// TIA Portal V19 export
FUNCTION "CEB_1" : Void   // FC14, LAD
{ S7_Optimized_Access := 'TRUE' }
// stored: SetENOAutomatically false
BEGIN

REGION Network 1: CEB_1 START
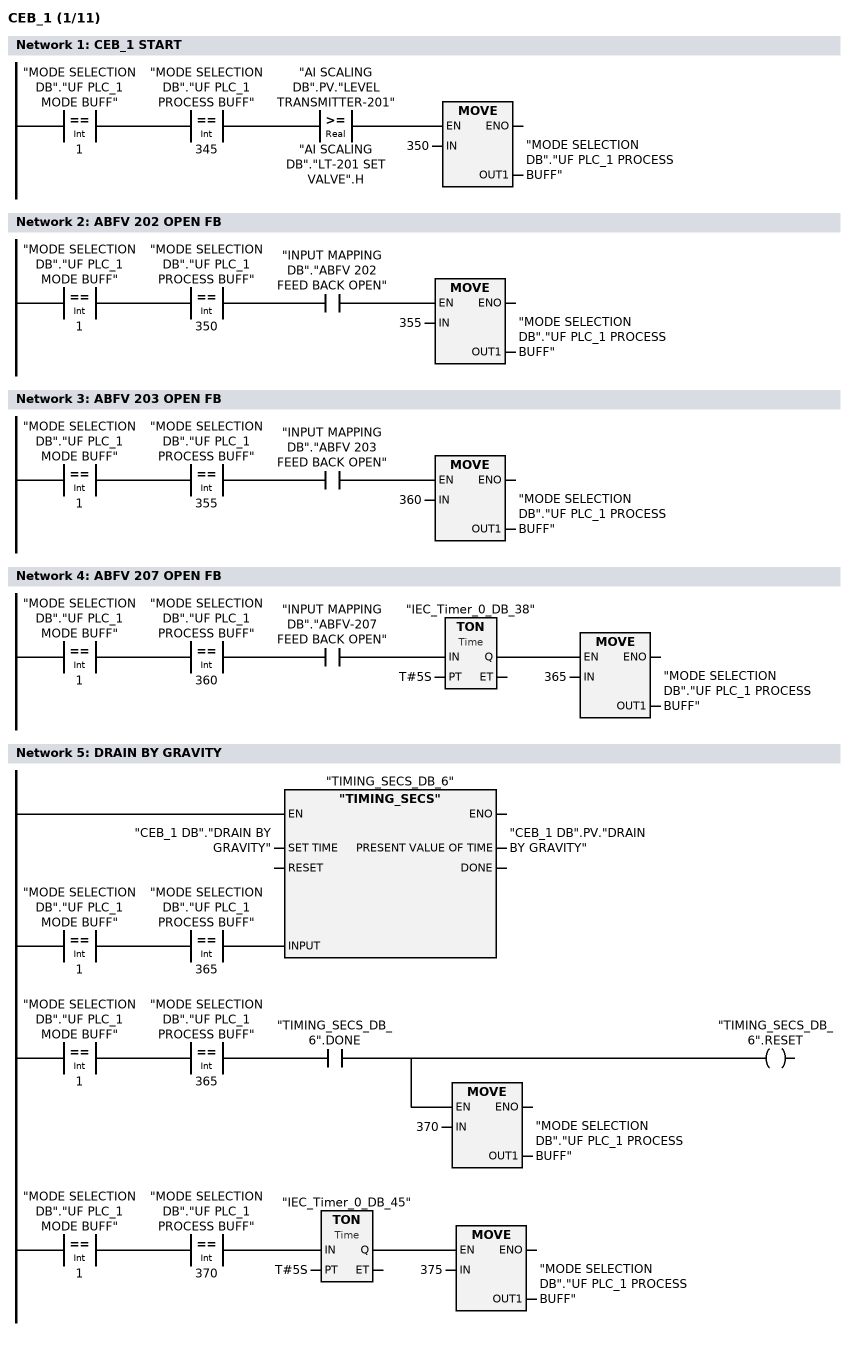
   RUNG wire#powerrail
      { S7_Templates := "SrcType := Int" } EQ_Contact(in1 := "MODE SELECTION DB"."UF PLC_1 MODE BUFF", in2 := 1)
      { S7_Templates := "SrcType := Int" } EQ_Contact(in1 := "MODE SELECTION DB"."UF PLC_1 PROCESS BUFF", in2 := 345)
      { S7_Templates := "SrcType := Real" } GE_Contact(in1 := "AI SCALING DB".PV."LEVEL TRANSMITTER-201", in2 := "AI SCALING DB"."LT-201 SET VALVE".H)
      Move(in := 350, out1 => "MODE SELECTION DB"."UF PLC_1 PROCESS BUFF")
   END_RUNG
   // the same network as SCL:
   IF ("MODE SELECTION DB"."UF PLC_1 MODE BUFF" = 1) AND ("MODE SELECTION DB"."UF PLC_1 PROCESS BUFF" = 345) AND ("AI SCALING DB".PV."LEVEL TRANSMITTER-201" >= "AI SCALING DB"."LT-201 SET VALVE".H) THEN
       "MODE SELECTION DB"."UF PLC_1 PROCESS BUFF" := 350;
   END_IF;
END_REGION

REGION Network 2: ABFV 202 OPEN FB
   RUNG wire#powerrail
      { S7_Templates := "SrcType := Int" } EQ_Contact(in1 := "MODE SELECTION DB"."UF PLC_1 MODE BUFF", in2 := 1)
      { S7_Templates := "SrcType := Int" } EQ_Contact(in1 := "MODE SELECTION DB"."UF PLC_1 PROCESS BUFF", in2 := 350)
      Contact( "INPUT MAPPING DB"."ABFV 202 FEED BACK OPEN" )
      Move(in := 355, out1 => "MODE SELECTION DB"."UF PLC_1 PROCESS BUFF")
   END_RUNG
   // the same network as SCL:
   IF ("MODE SELECTION DB"."UF PLC_1 MODE BUFF" = 1) AND ("MODE SELECTION DB"."UF PLC_1 PROCESS BUFF" = 350) AND "INPUT MAPPING DB"."ABFV 202 FEED BACK OPEN" THEN
       "MODE SELECTION DB"."UF PLC_1 PROCESS BUFF" := 355;
   END_IF;
END_REGION

REGION Network 3: ABFV 203 OPEN FB
   RUNG wire#powerrail
      { S7_Templates := "SrcType := Int" } EQ_Contact(in1 := "MODE SELECTION DB"."UF PLC_1 MODE BUFF", in2 := 1)
      { S7_Templates := "SrcType := Int" } EQ_Contact(in1 := "MODE SELECTION DB"."UF PLC_1 PROCESS BUFF", in2 := 355)
      Contact( "INPUT MAPPING DB"."ABFV 203 FEED BACK OPEN" )
      Move(in := 360, out1 => "MODE SELECTION DB"."UF PLC_1 PROCESS BUFF")
   END_RUNG
   // the same network as SCL:
   IF ("MODE SELECTION DB"."UF PLC_1 MODE BUFF" = 1) AND ("MODE SELECTION DB"."UF PLC_1 PROCESS BUFF" = 355) AND "INPUT MAPPING DB"."ABFV 203 FEED BACK OPEN" THEN
       "MODE SELECTION DB"."UF PLC_1 PROCESS BUFF" := 360;
   END_IF;
END_REGION

REGION Network 4: ABFV 207 OPEN FB
   RUNG wire#powerrail
      { S7_Templates := "SrcType := Int" } EQ_Contact(in1 := "MODE SELECTION DB"."UF PLC_1 MODE BUFF", in2 := 1)
      { S7_Templates := "SrcType := Int" } EQ_Contact(in1 := "MODE SELECTION DB"."UF PLC_1 PROCESS BUFF", in2 := 360)
      Contact( "INPUT MAPPING DB"."ABFV-207 FEED BACK OPEN" )
      { S7_Templates := "time_type := Time" } "IEC_Timer_0_DB_38".TON(pt := T#5S, et =>)
      Move(in := 365, out1 => "MODE SELECTION DB"."UF PLC_1 PROCESS BUFF")
   END_RUNG
   // the same network as SCL:
   "IEC_Timer_0_DB_38".TON(IN := ("MODE SELECTION DB"."UF PLC_1 MODE BUFF" = 1) AND ("MODE SELECTION DB"."UF PLC_1 PROCESS BUFF" = 360) AND "INPUT MAPPING DB"."ABFV-207 FEED BACK OPEN",
                           PT := T#5S);
   IF "IEC_Timer_0_DB_38".Q THEN "MODE SELECTION DB"."UF PLC_1 PROCESS BUFF" := 365; END_IF;
END_REGION

REGION Network 5: DRAIN BY GRAVITY
   RUNG wire#powerrail
      "TIMING_SECS_DB_6"(INPUT := wire#w1, "SET TIME" := "CEB_1 DB"."DRAIN BY GRAVITY", RESET :=, "PRESENT VALUE OF TIME" => "CEB_1 DB".PV."DRAIN BY GRAVITY", DONE =>)
   END_RUNG
   RUNG wire#powerrail
      { S7_Templates := "SrcType := Int" } EQ_Contact(in1 := "MODE SELECTION DB"."UF PLC_1 MODE BUFF", in2 := 1)
      { S7_Templates := "SrcType := Int" } EQ_Contact(in1 := "MODE SELECTION DB"."UF PLC_1 PROCESS BUFF", in2 := 365)
   END_RUNG wire#w1
   RUNG wire#powerrail
      { S7_Templates := "SrcType := Int" } EQ_Contact(in1 := "MODE SELECTION DB"."UF PLC_1 MODE BUFF", in2 := 1)
      { S7_Templates := "SrcType := Int" } EQ_Contact(in1 := "MODE SELECTION DB"."UF PLC_1 PROCESS BUFF", in2 := 365)
      Contact( "TIMING_SECS_DB_6".DONE )
      wire#w2
      Coil( "TIMING_SECS_DB_6".RESET )
   END_RUNG
   RUNG wire#w2
      Move(in := 370, out1 => "MODE SELECTION DB"."UF PLC_1 PROCESS BUFF")
   END_RUNG
   RUNG wire#powerrail
      { S7_Templates := "SrcType := Int" } EQ_Contact(in1 := "MODE SELECTION DB"."UF PLC_1 MODE BUFF", in2 := 1)
      { S7_Templates := "SrcType := Int" } EQ_Contact(in1 := "MODE SELECTION DB"."UF PLC_1 PROCESS BUFF", in2 := 370)
      { S7_Templates := "time_type := Time" } "IEC_Timer_0_DB_45".TON(pt := T#5S, et =>)
      Move(in := 375, out1 => "MODE SELECTION DB"."UF PLC_1 PROCESS BUFF")
   END_RUNG
   // the same network as SCL:
   "TIMING_SECS_DB_6"("SET TIME" := "CEB_1 DB"."DRAIN BY GRAVITY",   // "TIMING_SECS"
                      INPUT := ("MODE SELECTION DB"."UF PLC_1 MODE BUFF" = 1) AND ("MODE SELECTION DB"."UF PLC_1 PROCESS BUFF" = 365),
                      "PRESENT VALUE OF TIME" => "CEB_1 DB".PV."DRAIN BY GRAVITY");
   "TIMING_SECS_DB_6".RESET := ("MODE SELECTION DB"."UF PLC_1 MODE BUFF" = 1) AND ("MODE SELECTION DB"."UF PLC_1 PROCESS BUFF" = 365) AND "TIMING_SECS_DB_6".DONE;
   IF "TIMING_SECS_DB_6".RESET THEN "MODE SELECTION DB"."UF PLC_1 PROCESS BUFF" := 370; END_IF;
   "IEC_Timer_0_DB_45".TON(IN := ("MODE SELECTION DB"."UF PLC_1 MODE BUFF" = 1) AND ("MODE SELECTION DB"."UF PLC_1 PROCESS BUFF" = 370),
                           PT := T#5S);
   IF "IEC_Timer_0_DB_45".Q THEN "MODE SELECTION DB"."UF PLC_1 PROCESS BUFF" := 375; END_IF;
END_REGION

REGION Network 6: ABFV 207 CLOSE FB
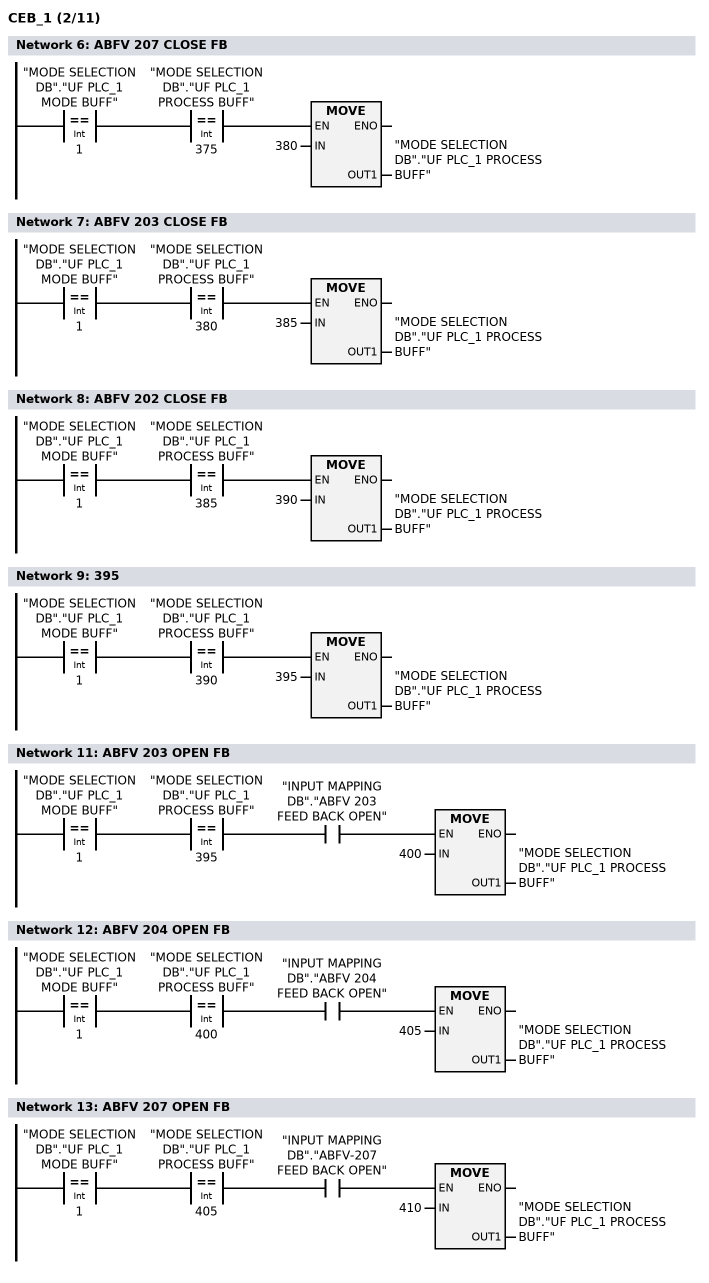
   RUNG wire#powerrail
      { S7_Templates := "SrcType := Int" } EQ_Contact(in1 := "MODE SELECTION DB"."UF PLC_1 MODE BUFF", in2 := 1)
      { S7_Templates := "SrcType := Int" } EQ_Contact(in1 := "MODE SELECTION DB"."UF PLC_1 PROCESS BUFF", in2 := 375)
      Move(in := 380, out1 => "MODE SELECTION DB"."UF PLC_1 PROCESS BUFF")
   END_RUNG
   // the same network as SCL:
   IF ("MODE SELECTION DB"."UF PLC_1 MODE BUFF" = 1) AND ("MODE SELECTION DB"."UF PLC_1 PROCESS BUFF" = 375) THEN
       "MODE SELECTION DB"."UF PLC_1 PROCESS BUFF" := 380;
   END_IF;
END_REGION

REGION Network 7: ABFV 203 CLOSE FB
   RUNG wire#powerrail
      { S7_Templates := "SrcType := Int" } EQ_Contact(in1 := "MODE SELECTION DB"."UF PLC_1 MODE BUFF", in2 := 1)
      { S7_Templates := "SrcType := Int" } EQ_Contact(in1 := "MODE SELECTION DB"."UF PLC_1 PROCESS BUFF", in2 := 380)
      Move(in := 385, out1 => "MODE SELECTION DB"."UF PLC_1 PROCESS BUFF")
   END_RUNG
   // the same network as SCL:
   IF ("MODE SELECTION DB"."UF PLC_1 MODE BUFF" = 1) AND ("MODE SELECTION DB"."UF PLC_1 PROCESS BUFF" = 380) THEN
       "MODE SELECTION DB"."UF PLC_1 PROCESS BUFF" := 385;
   END_IF;
END_REGION

REGION Network 8: ABFV 202 CLOSE FB
   RUNG wire#powerrail
      { S7_Templates := "SrcType := Int" } EQ_Contact(in1 := "MODE SELECTION DB"."UF PLC_1 MODE BUFF", in2 := 1)
      { S7_Templates := "SrcType := Int" } EQ_Contact(in1 := "MODE SELECTION DB"."UF PLC_1 PROCESS BUFF", in2 := 385)
      Move(in := 390, out1 => "MODE SELECTION DB"."UF PLC_1 PROCESS BUFF")
   END_RUNG
   // the same network as SCL:
   IF ("MODE SELECTION DB"."UF PLC_1 MODE BUFF" = 1) AND ("MODE SELECTION DB"."UF PLC_1 PROCESS BUFF" = 385) THEN
       "MODE SELECTION DB"."UF PLC_1 PROCESS BUFF" := 390;
   END_IF;
END_REGION

REGION Network 9: 395
   RUNG wire#powerrail
      { S7_Templates := "SrcType := Int" } EQ_Contact(in1 := "MODE SELECTION DB"."UF PLC_1 MODE BUFF", in2 := 1)
      { S7_Templates := "SrcType := Int" } EQ_Contact(in1 := "MODE SELECTION DB"."UF PLC_1 PROCESS BUFF", in2 := 390)
      Move(in := 395, out1 => "MODE SELECTION DB"."UF PLC_1 PROCESS BUFF")
   END_RUNG
   // the same network as SCL:
   IF ("MODE SELECTION DB"."UF PLC_1 MODE BUFF" = 1) AND ("MODE SELECTION DB"."UF PLC_1 PROCESS BUFF" = 390) THEN
       "MODE SELECTION DB"."UF PLC_1 PROCESS BUFF" := 395;
   END_IF;
END_REGION

REGION Network 11: ABFV 203 OPEN FB
   RUNG wire#powerrail
      { S7_Templates := "SrcType := Int" } EQ_Contact(in1 := "MODE SELECTION DB"."UF PLC_1 MODE BUFF", in2 := 1)
      { S7_Templates := "SrcType := Int" } EQ_Contact(in1 := "MODE SELECTION DB"."UF PLC_1 PROCESS BUFF", in2 := 395)
      Contact( "INPUT MAPPING DB"."ABFV 203 FEED BACK OPEN" )
      Move(in := 400, out1 => "MODE SELECTION DB"."UF PLC_1 PROCESS BUFF")
   END_RUNG
   // the same network as SCL:
   IF ("MODE SELECTION DB"."UF PLC_1 MODE BUFF" = 1) AND ("MODE SELECTION DB"."UF PLC_1 PROCESS BUFF" = 395) AND "INPUT MAPPING DB"."ABFV 203 FEED BACK OPEN" THEN
       "MODE SELECTION DB"."UF PLC_1 PROCESS BUFF" := 400;
   END_IF;
END_REGION

REGION Network 12: ABFV 204 OPEN FB
   RUNG wire#powerrail
      { S7_Templates := "SrcType := Int" } EQ_Contact(in1 := "MODE SELECTION DB"."UF PLC_1 MODE BUFF", in2 := 1)
      { S7_Templates := "SrcType := Int" } EQ_Contact(in1 := "MODE SELECTION DB"."UF PLC_1 PROCESS BUFF", in2 := 400)
      Contact( "INPUT MAPPING DB"."ABFV 204 FEED BACK OPEN" )
      Move(in := 405, out1 => "MODE SELECTION DB"."UF PLC_1 PROCESS BUFF")
   END_RUNG
   // the same network as SCL:
   IF ("MODE SELECTION DB"."UF PLC_1 MODE BUFF" = 1) AND ("MODE SELECTION DB"."UF PLC_1 PROCESS BUFF" = 400) AND "INPUT MAPPING DB"."ABFV 204 FEED BACK OPEN" THEN
       "MODE SELECTION DB"."UF PLC_1 PROCESS BUFF" := 405;
   END_IF;
END_REGION

REGION Network 13: ABFV 207 OPEN FB
   RUNG wire#powerrail
      { S7_Templates := "SrcType := Int" } EQ_Contact(in1 := "MODE SELECTION DB"."UF PLC_1 MODE BUFF", in2 := 1)
      { S7_Templates := "SrcType := Int" } EQ_Contact(in1 := "MODE SELECTION DB"."UF PLC_1 PROCESS BUFF", in2 := 405)
      Contact( "INPUT MAPPING DB"."ABFV-207 FEED BACK OPEN" )
      Move(in := 410, out1 => "MODE SELECTION DB"."UF PLC_1 PROCESS BUFF")
   END_RUNG
   // the same network as SCL:
   IF ("MODE SELECTION DB"."UF PLC_1 MODE BUFF" = 1) AND ("MODE SELECTION DB"."UF PLC_1 PROCESS BUFF" = 405) AND "INPUT MAPPING DB"."ABFV-207 FEED BACK OPEN" THEN
       "MODE SELECTION DB"."UF PLC_1 PROCESS BUFF" := 410;
   END_IF;
END_REGION

REGION Network 14: ABFV 208 OPEN FB
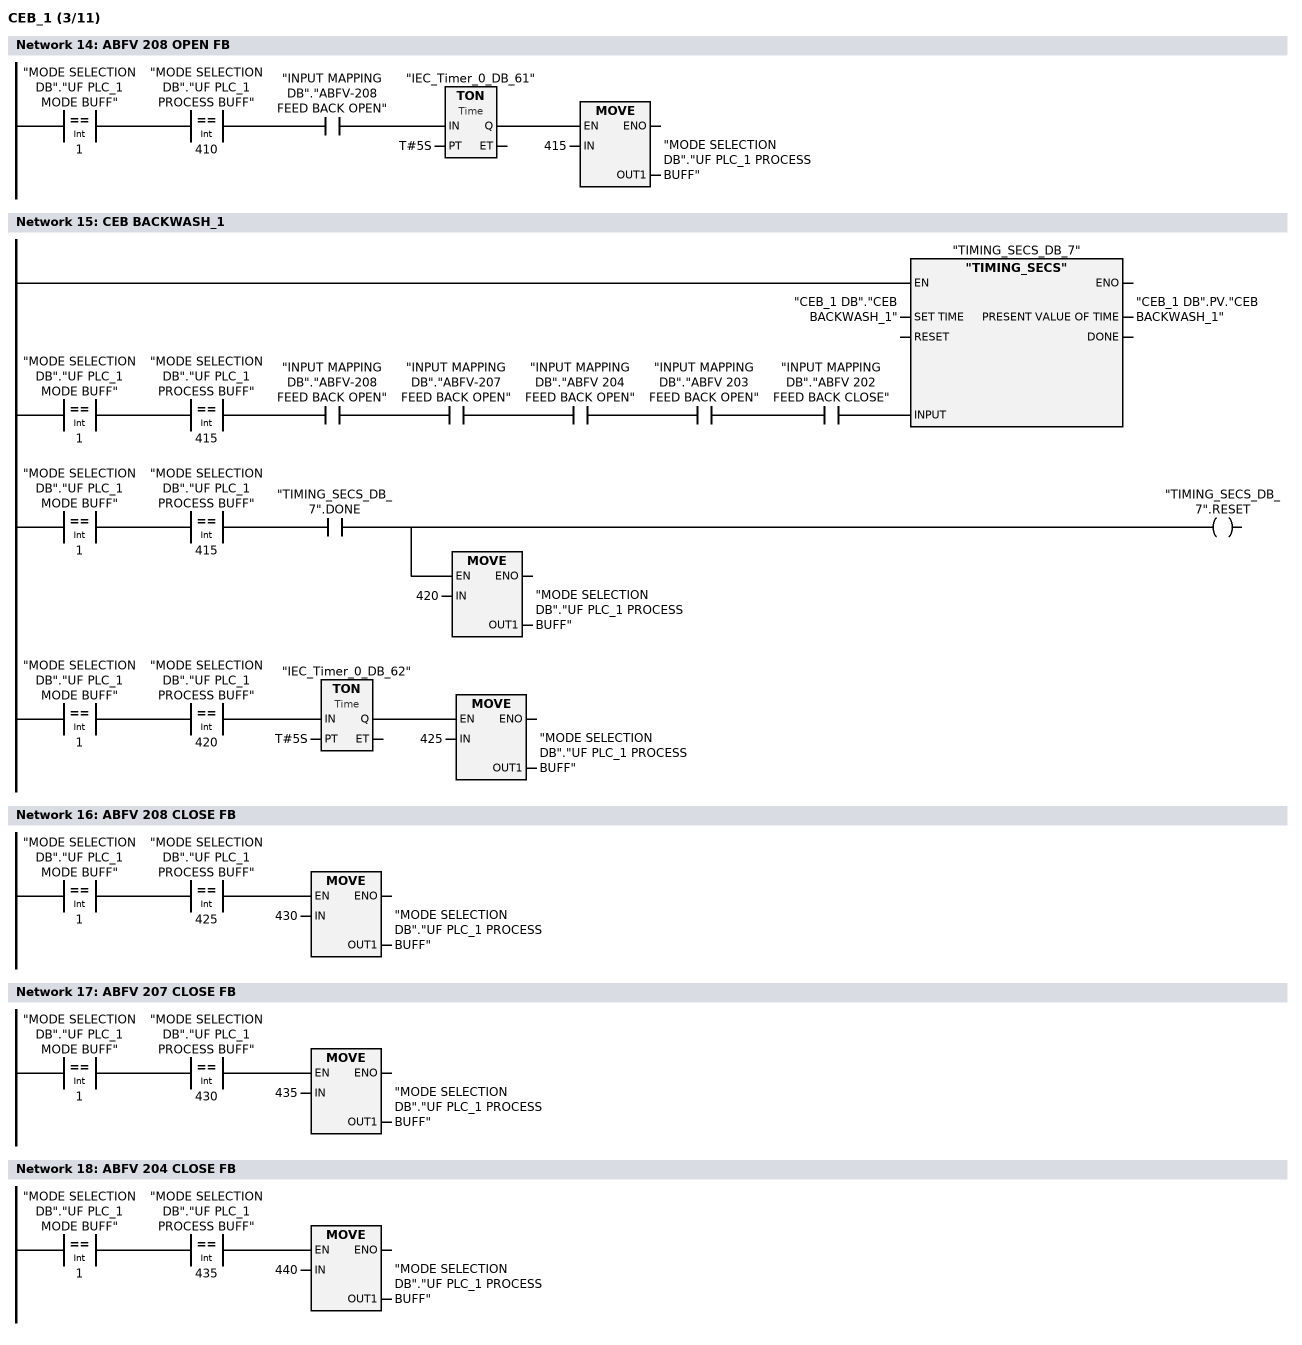
   RUNG wire#powerrail
      { S7_Templates := "SrcType := Int" } EQ_Contact(in1 := "MODE SELECTION DB"."UF PLC_1 MODE BUFF", in2 := 1)
      { S7_Templates := "SrcType := Int" } EQ_Contact(in1 := "MODE SELECTION DB"."UF PLC_1 PROCESS BUFF", in2 := 410)
      Contact( "INPUT MAPPING DB"."ABFV-208 FEED BACK OPEN" )
      { S7_Templates := "time_type := Time" } "IEC_Timer_0_DB_61".TON(pt := T#5S, et =>)
      Move(in := 415, out1 => "MODE SELECTION DB"."UF PLC_1 PROCESS BUFF")
   END_RUNG
   // the same network as SCL:
   "IEC_Timer_0_DB_61".TON(IN := ("MODE SELECTION DB"."UF PLC_1 MODE BUFF" = 1) AND ("MODE SELECTION DB"."UF PLC_1 PROCESS BUFF" = 410) AND "INPUT MAPPING DB"."ABFV-208 FEED BACK OPEN",
                           PT := T#5S);
   IF "IEC_Timer_0_DB_61".Q THEN "MODE SELECTION DB"."UF PLC_1 PROCESS BUFF" := 415; END_IF;
END_REGION

REGION Network 15: CEB BACKWASH_1
   RUNG wire#powerrail
      "TIMING_SECS_DB_7"(INPUT := wire#w1, "SET TIME" := "CEB_1 DB"."CEB BACKWASH_1", RESET :=, "PRESENT VALUE OF TIME" => "CEB_1 DB".PV."CEB BACKWASH_1", DONE =>)
   END_RUNG
   RUNG wire#powerrail
      { S7_Templates := "SrcType := Int" } EQ_Contact(in1 := "MODE SELECTION DB"."UF PLC_1 MODE BUFF", in2 := 1)
      { S7_Templates := "SrcType := Int" } EQ_Contact(in1 := "MODE SELECTION DB"."UF PLC_1 PROCESS BUFF", in2 := 415)
      Contact( "INPUT MAPPING DB"."ABFV-208 FEED BACK OPEN" )
      Contact( "INPUT MAPPING DB"."ABFV-207 FEED BACK OPEN" )
      Contact( "INPUT MAPPING DB"."ABFV 204 FEED BACK OPEN" )
      Contact( "INPUT MAPPING DB"."ABFV 203 FEED BACK OPEN" )
      Contact( "INPUT MAPPING DB"."ABFV 202 FEED BACK CLOSE" )
   END_RUNG wire#w1
   RUNG wire#powerrail
      { S7_Templates := "SrcType := Int" } EQ_Contact(in1 := "MODE SELECTION DB"."UF PLC_1 MODE BUFF", in2 := 1)
      { S7_Templates := "SrcType := Int" } EQ_Contact(in1 := "MODE SELECTION DB"."UF PLC_1 PROCESS BUFF", in2 := 415)
      Contact( "TIMING_SECS_DB_7".DONE )
      wire#w2
      Coil( "TIMING_SECS_DB_7".RESET )
   END_RUNG
   RUNG wire#w2
      Move(in := 420, out1 => "MODE SELECTION DB"."UF PLC_1 PROCESS BUFF")
   END_RUNG
   RUNG wire#powerrail
      { S7_Templates := "SrcType := Int" } EQ_Contact(in1 := "MODE SELECTION DB"."UF PLC_1 MODE BUFF", in2 := 1)
      { S7_Templates := "SrcType := Int" } EQ_Contact(in1 := "MODE SELECTION DB"."UF PLC_1 PROCESS BUFF", in2 := 420)
      { S7_Templates := "time_type := Time" } "IEC_Timer_0_DB_62".TON(pt := T#5S, et =>)
      Move(in := 425, out1 => "MODE SELECTION DB"."UF PLC_1 PROCESS BUFF")
   END_RUNG
   // the same network as SCL:
   "TIMING_SECS_DB_7"("SET TIME" := "CEB_1 DB"."CEB BACKWASH_1",   // "TIMING_SECS"
                      INPUT := ("MODE SELECTION DB"."UF PLC_1 MODE BUFF" = 1) AND ("MODE SELECTION DB"."UF PLC_1 PROCESS BUFF" = 415) AND "INPUT MAPPING DB"."ABFV-208 FEED BACK OPEN" AND "INPUT MAPPING DB"."ABFV-207 FEED BACK OPEN" AND "INPUT MAPPING DB"."ABFV 204 FEED BACK OPEN" AND "INPUT MAPPING DB"."ABFV 203 FEED BACK OPEN" AND "INPUT MAPPING DB"."ABFV 202 FEED BACK CLOSE",
                      "PRESENT VALUE OF TIME" => "CEB_1 DB".PV."CEB BACKWASH_1");
   "TIMING_SECS_DB_7".RESET := ("MODE SELECTION DB"."UF PLC_1 MODE BUFF" = 1) AND ("MODE SELECTION DB"."UF PLC_1 PROCESS BUFF" = 415) AND "TIMING_SECS_DB_7".DONE;
   IF "TIMING_SECS_DB_7".RESET THEN "MODE SELECTION DB"."UF PLC_1 PROCESS BUFF" := 420; END_IF;
   "IEC_Timer_0_DB_62".TON(IN := ("MODE SELECTION DB"."UF PLC_1 MODE BUFF" = 1) AND ("MODE SELECTION DB"."UF PLC_1 PROCESS BUFF" = 420),
                           PT := T#5S);
   IF "IEC_Timer_0_DB_62".Q THEN "MODE SELECTION DB"."UF PLC_1 PROCESS BUFF" := 425; END_IF;
END_REGION

REGION Network 16: ABFV 208 CLOSE FB
   RUNG wire#powerrail
      { S7_Templates := "SrcType := Int" } EQ_Contact(in1 := "MODE SELECTION DB"."UF PLC_1 MODE BUFF", in2 := 1)
      { S7_Templates := "SrcType := Int" } EQ_Contact(in1 := "MODE SELECTION DB"."UF PLC_1 PROCESS BUFF", in2 := 425)
      Move(in := 430, out1 => "MODE SELECTION DB"."UF PLC_1 PROCESS BUFF")
   END_RUNG
   // the same network as SCL:
   IF ("MODE SELECTION DB"."UF PLC_1 MODE BUFF" = 1) AND ("MODE SELECTION DB"."UF PLC_1 PROCESS BUFF" = 425) THEN
       "MODE SELECTION DB"."UF PLC_1 PROCESS BUFF" := 430;
   END_IF;
END_REGION

REGION Network 17: ABFV 207 CLOSE FB
   RUNG wire#powerrail
      { S7_Templates := "SrcType := Int" } EQ_Contact(in1 := "MODE SELECTION DB"."UF PLC_1 MODE BUFF", in2 := 1)
      { S7_Templates := "SrcType := Int" } EQ_Contact(in1 := "MODE SELECTION DB"."UF PLC_1 PROCESS BUFF", in2 := 430)
      Move(in := 435, out1 => "MODE SELECTION DB"."UF PLC_1 PROCESS BUFF")
   END_RUNG
   // the same network as SCL:
   IF ("MODE SELECTION DB"."UF PLC_1 MODE BUFF" = 1) AND ("MODE SELECTION DB"."UF PLC_1 PROCESS BUFF" = 430) THEN
       "MODE SELECTION DB"."UF PLC_1 PROCESS BUFF" := 435;
   END_IF;
END_REGION

REGION Network 18: ABFV 204 CLOSE FB
   RUNG wire#powerrail
      { S7_Templates := "SrcType := Int" } EQ_Contact(in1 := "MODE SELECTION DB"."UF PLC_1 MODE BUFF", in2 := 1)
      { S7_Templates := "SrcType := Int" } EQ_Contact(in1 := "MODE SELECTION DB"."UF PLC_1 PROCESS BUFF", in2 := 435)
      Move(in := 440, out1 => "MODE SELECTION DB"."UF PLC_1 PROCESS BUFF")
   END_RUNG
   // the same network as SCL:
   IF ("MODE SELECTION DB"."UF PLC_1 MODE BUFF" = 1) AND ("MODE SELECTION DB"."UF PLC_1 PROCESS BUFF" = 435) THEN
       "MODE SELECTION DB"."UF PLC_1 PROCESS BUFF" := 440;
   END_IF;
END_REGION

REGION Network 19: ABFV 203 CLOSE FB
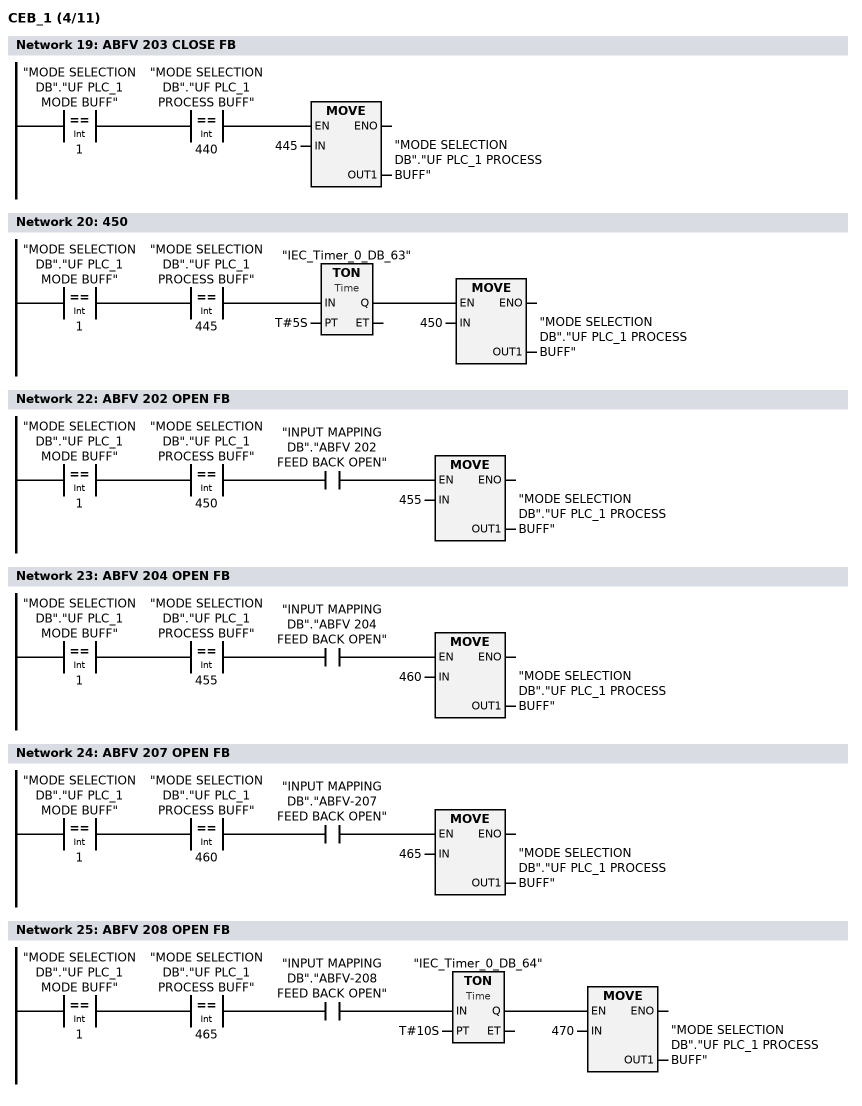
   RUNG wire#powerrail
      { S7_Templates := "SrcType := Int" } EQ_Contact(in1 := "MODE SELECTION DB"."UF PLC_1 MODE BUFF", in2 := 1)
      { S7_Templates := "SrcType := Int" } EQ_Contact(in1 := "MODE SELECTION DB"."UF PLC_1 PROCESS BUFF", in2 := 440)
      Move(in := 445, out1 => "MODE SELECTION DB"."UF PLC_1 PROCESS BUFF")
   END_RUNG
   // the same network as SCL:
   IF ("MODE SELECTION DB"."UF PLC_1 MODE BUFF" = 1) AND ("MODE SELECTION DB"."UF PLC_1 PROCESS BUFF" = 440) THEN
       "MODE SELECTION DB"."UF PLC_1 PROCESS BUFF" := 445;
   END_IF;
END_REGION

REGION Network 20: 450
   RUNG wire#powerrail
      { S7_Templates := "SrcType := Int" } EQ_Contact(in1 := "MODE SELECTION DB"."UF PLC_1 MODE BUFF", in2 := 1)
      { S7_Templates := "SrcType := Int" } EQ_Contact(in1 := "MODE SELECTION DB"."UF PLC_1 PROCESS BUFF", in2 := 445)
      { S7_Templates := "time_type := Time" } "IEC_Timer_0_DB_63".TON(pt := T#5S, et =>)
      Move(in := 450, out1 => "MODE SELECTION DB"."UF PLC_1 PROCESS BUFF")
   END_RUNG
   // the same network as SCL:
   "IEC_Timer_0_DB_63".TON(IN := ("MODE SELECTION DB"."UF PLC_1 MODE BUFF" = 1) AND ("MODE SELECTION DB"."UF PLC_1 PROCESS BUFF" = 445),
                           PT := T#5S);
   IF "IEC_Timer_0_DB_63".Q THEN "MODE SELECTION DB"."UF PLC_1 PROCESS BUFF" := 450; END_IF;
END_REGION

REGION Network 22: ABFV 202 OPEN FB
   RUNG wire#powerrail
      { S7_Templates := "SrcType := Int" } EQ_Contact(in1 := "MODE SELECTION DB"."UF PLC_1 MODE BUFF", in2 := 1)
      { S7_Templates := "SrcType := Int" } EQ_Contact(in1 := "MODE SELECTION DB"."UF PLC_1 PROCESS BUFF", in2 := 450)
      Contact( "INPUT MAPPING DB"."ABFV 202 FEED BACK OPEN" )
      Move(in := 455, out1 => "MODE SELECTION DB"."UF PLC_1 PROCESS BUFF")
   END_RUNG
   // the same network as SCL:
   IF ("MODE SELECTION DB"."UF PLC_1 MODE BUFF" = 1) AND ("MODE SELECTION DB"."UF PLC_1 PROCESS BUFF" = 450) AND "INPUT MAPPING DB"."ABFV 202 FEED BACK OPEN" THEN
       "MODE SELECTION DB"."UF PLC_1 PROCESS BUFF" := 455;
   END_IF;
END_REGION

REGION Network 23: ABFV 204 OPEN FB
   RUNG wire#powerrail
      { S7_Templates := "SrcType := Int" } EQ_Contact(in1 := "MODE SELECTION DB"."UF PLC_1 MODE BUFF", in2 := 1)
      { S7_Templates := "SrcType := Int" } EQ_Contact(in1 := "MODE SELECTION DB"."UF PLC_1 PROCESS BUFF", in2 := 455)
      Contact( "INPUT MAPPING DB"."ABFV 204 FEED BACK OPEN" )
      Move(in := 460, out1 => "MODE SELECTION DB"."UF PLC_1 PROCESS BUFF")
   END_RUNG
   // the same network as SCL:
   IF ("MODE SELECTION DB"."UF PLC_1 MODE BUFF" = 1) AND ("MODE SELECTION DB"."UF PLC_1 PROCESS BUFF" = 455) AND "INPUT MAPPING DB"."ABFV 204 FEED BACK OPEN" THEN
       "MODE SELECTION DB"."UF PLC_1 PROCESS BUFF" := 460;
   END_IF;
END_REGION

REGION Network 24: ABFV 207 OPEN FB
   RUNG wire#powerrail
      { S7_Templates := "SrcType := Int" } EQ_Contact(in1 := "MODE SELECTION DB"."UF PLC_1 MODE BUFF", in2 := 1)
      { S7_Templates := "SrcType := Int" } EQ_Contact(in1 := "MODE SELECTION DB"."UF PLC_1 PROCESS BUFF", in2 := 460)
      Contact( "INPUT MAPPING DB"."ABFV-207 FEED BACK OPEN" )
      Move(in := 465, out1 => "MODE SELECTION DB"."UF PLC_1 PROCESS BUFF")
   END_RUNG
   // the same network as SCL:
   IF ("MODE SELECTION DB"."UF PLC_1 MODE BUFF" = 1) AND ("MODE SELECTION DB"."UF PLC_1 PROCESS BUFF" = 460) AND "INPUT MAPPING DB"."ABFV-207 FEED BACK OPEN" THEN
       "MODE SELECTION DB"."UF PLC_1 PROCESS BUFF" := 465;
   END_IF;
END_REGION

REGION Network 25: ABFV 208 OPEN FB
   RUNG wire#powerrail
      { S7_Templates := "SrcType := Int" } EQ_Contact(in1 := "MODE SELECTION DB"."UF PLC_1 MODE BUFF", in2 := 1)
      { S7_Templates := "SrcType := Int" } EQ_Contact(in1 := "MODE SELECTION DB"."UF PLC_1 PROCESS BUFF", in2 := 465)
      Contact( "INPUT MAPPING DB"."ABFV-208 FEED BACK OPEN" )
      { S7_Templates := "time_type := Time" } "IEC_Timer_0_DB_64".TON(pt := T#10S, et =>)
      Move(in := 470, out1 => "MODE SELECTION DB"."UF PLC_1 PROCESS BUFF")
   END_RUNG
   // the same network as SCL:
   "IEC_Timer_0_DB_64".TON(IN := ("MODE SELECTION DB"."UF PLC_1 MODE BUFF" = 1) AND ("MODE SELECTION DB"."UF PLC_1 PROCESS BUFF" = 465) AND "INPUT MAPPING DB"."ABFV-208 FEED BACK OPEN",
                           PT := T#10S);
   IF "IEC_Timer_0_DB_64".Q THEN "MODE SELECTION DB"."UF PLC_1 PROCESS BUFF" := 470; END_IF;
END_REGION

REGION Network 26: CEB BACKWASH_2
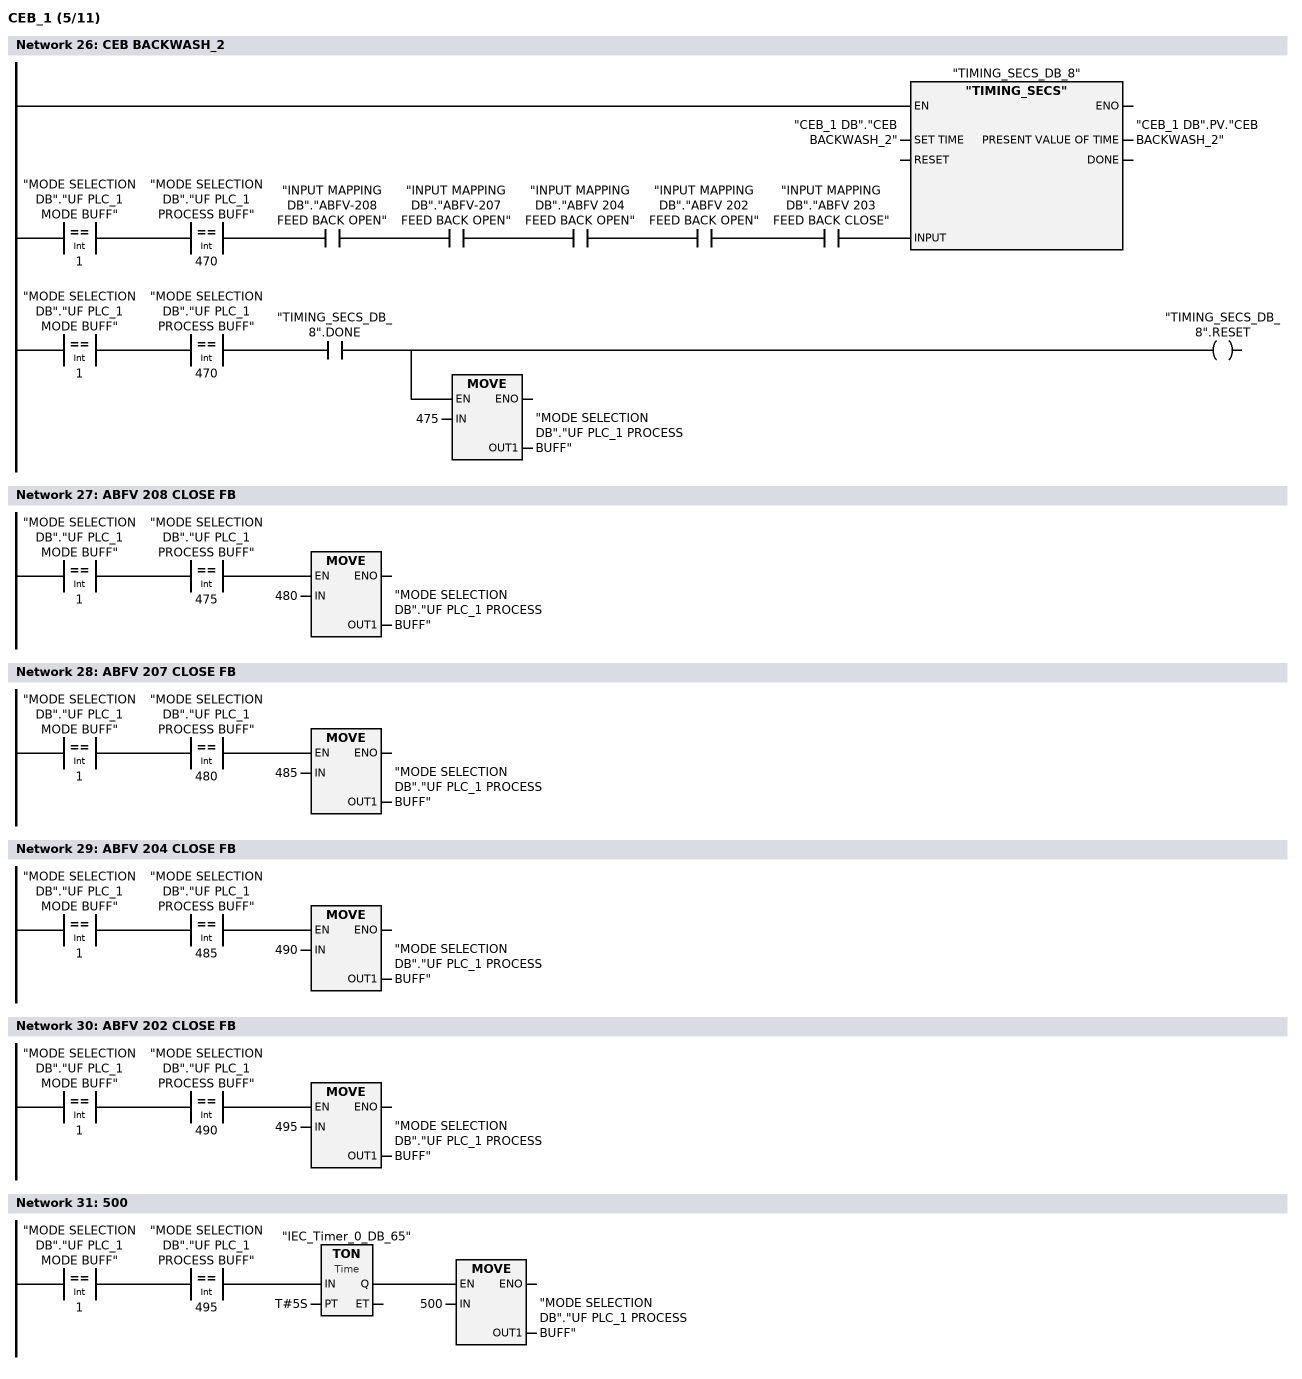
   RUNG wire#powerrail
      "TIMING_SECS_DB_8"(INPUT := wire#w1, "SET TIME" := "CEB_1 DB"."CEB BACKWASH_2", RESET :=, "PRESENT VALUE OF TIME" => "CEB_1 DB".PV."CEB BACKWASH_2", DONE =>)
   END_RUNG
   RUNG wire#powerrail
      { S7_Templates := "SrcType := Int" } EQ_Contact(in1 := "MODE SELECTION DB"."UF PLC_1 MODE BUFF", in2 := 1)
      { S7_Templates := "SrcType := Int" } EQ_Contact(in1 := "MODE SELECTION DB"."UF PLC_1 PROCESS BUFF", in2 := 470)
      Contact( "INPUT MAPPING DB"."ABFV-208 FEED BACK OPEN" )
      Contact( "INPUT MAPPING DB"."ABFV-207 FEED BACK OPEN" )
      Contact( "INPUT MAPPING DB"."ABFV 204 FEED BACK OPEN" )
      Contact( "INPUT MAPPING DB"."ABFV 202 FEED BACK OPEN" )
      Contact( "INPUT MAPPING DB"."ABFV 203 FEED BACK CLOSE" )
   END_RUNG wire#w1
   RUNG wire#powerrail
      { S7_Templates := "SrcType := Int" } EQ_Contact(in1 := "MODE SELECTION DB"."UF PLC_1 MODE BUFF", in2 := 1)
      { S7_Templates := "SrcType := Int" } EQ_Contact(in1 := "MODE SELECTION DB"."UF PLC_1 PROCESS BUFF", in2 := 470)
      Contact( "TIMING_SECS_DB_8".DONE )
      wire#w2
      Coil( "TIMING_SECS_DB_8".RESET )
   END_RUNG
   RUNG wire#w2
      Move(in := 475, out1 => "MODE SELECTION DB"."UF PLC_1 PROCESS BUFF")
   END_RUNG
   // the same network as SCL:
   "TIMING_SECS_DB_8"("SET TIME" := "CEB_1 DB"."CEB BACKWASH_2",   // "TIMING_SECS"
                      INPUT := ("MODE SELECTION DB"."UF PLC_1 MODE BUFF" = 1) AND ("MODE SELECTION DB"."UF PLC_1 PROCESS BUFF" = 470) AND "INPUT MAPPING DB"."ABFV-208 FEED BACK OPEN" AND "INPUT MAPPING DB"."ABFV-207 FEED BACK OPEN" AND "INPUT MAPPING DB"."ABFV 204 FEED BACK OPEN" AND "INPUT MAPPING DB"."ABFV 202 FEED BACK OPEN" AND "INPUT MAPPING DB"."ABFV 203 FEED BACK CLOSE",
                      "PRESENT VALUE OF TIME" => "CEB_1 DB".PV."CEB BACKWASH_2");
   "TIMING_SECS_DB_8".RESET := ("MODE SELECTION DB"."UF PLC_1 MODE BUFF" = 1) AND ("MODE SELECTION DB"."UF PLC_1 PROCESS BUFF" = 470) AND "TIMING_SECS_DB_8".DONE;
   IF "TIMING_SECS_DB_8".RESET THEN "MODE SELECTION DB"."UF PLC_1 PROCESS BUFF" := 475; END_IF;
END_REGION

REGION Network 27: ABFV 208 CLOSE FB
   RUNG wire#powerrail
      { S7_Templates := "SrcType := Int" } EQ_Contact(in1 := "MODE SELECTION DB"."UF PLC_1 MODE BUFF", in2 := 1)
      { S7_Templates := "SrcType := Int" } EQ_Contact(in1 := "MODE SELECTION DB"."UF PLC_1 PROCESS BUFF", in2 := 475)
      Move(in := 480, out1 => "MODE SELECTION DB"."UF PLC_1 PROCESS BUFF")
   END_RUNG
   // the same network as SCL:
   IF ("MODE SELECTION DB"."UF PLC_1 MODE BUFF" = 1) AND ("MODE SELECTION DB"."UF PLC_1 PROCESS BUFF" = 475) THEN
       "MODE SELECTION DB"."UF PLC_1 PROCESS BUFF" := 480;
   END_IF;
END_REGION

REGION Network 28: ABFV 207 CLOSE FB
   RUNG wire#powerrail
      { S7_Templates := "SrcType := Int" } EQ_Contact(in1 := "MODE SELECTION DB"."UF PLC_1 MODE BUFF", in2 := 1)
      { S7_Templates := "SrcType := Int" } EQ_Contact(in1 := "MODE SELECTION DB"."UF PLC_1 PROCESS BUFF", in2 := 480)
      Move(in := 485, out1 => "MODE SELECTION DB"."UF PLC_1 PROCESS BUFF")
   END_RUNG
   // the same network as SCL:
   IF ("MODE SELECTION DB"."UF PLC_1 MODE BUFF" = 1) AND ("MODE SELECTION DB"."UF PLC_1 PROCESS BUFF" = 480) THEN
       "MODE SELECTION DB"."UF PLC_1 PROCESS BUFF" := 485;
   END_IF;
END_REGION

REGION Network 29: ABFV 204 CLOSE FB
   RUNG wire#powerrail
      { S7_Templates := "SrcType := Int" } EQ_Contact(in1 := "MODE SELECTION DB"."UF PLC_1 MODE BUFF", in2 := 1)
      { S7_Templates := "SrcType := Int" } EQ_Contact(in1 := "MODE SELECTION DB"."UF PLC_1 PROCESS BUFF", in2 := 485)
      Move(in := 490, out1 => "MODE SELECTION DB"."UF PLC_1 PROCESS BUFF")
   END_RUNG
   // the same network as SCL:
   IF ("MODE SELECTION DB"."UF PLC_1 MODE BUFF" = 1) AND ("MODE SELECTION DB"."UF PLC_1 PROCESS BUFF" = 485) THEN
       "MODE SELECTION DB"."UF PLC_1 PROCESS BUFF" := 490;
   END_IF;
END_REGION

REGION Network 30: ABFV 202 CLOSE FB
   RUNG wire#powerrail
      { S7_Templates := "SrcType := Int" } EQ_Contact(in1 := "MODE SELECTION DB"."UF PLC_1 MODE BUFF", in2 := 1)
      { S7_Templates := "SrcType := Int" } EQ_Contact(in1 := "MODE SELECTION DB"."UF PLC_1 PROCESS BUFF", in2 := 490)
      Move(in := 495, out1 => "MODE SELECTION DB"."UF PLC_1 PROCESS BUFF")
   END_RUNG
   // the same network as SCL:
   IF ("MODE SELECTION DB"."UF PLC_1 MODE BUFF" = 1) AND ("MODE SELECTION DB"."UF PLC_1 PROCESS BUFF" = 490) THEN
       "MODE SELECTION DB"."UF PLC_1 PROCESS BUFF" := 495;
   END_IF;
END_REGION

REGION Network 31: 500
   RUNG wire#powerrail
      { S7_Templates := "SrcType := Int" } EQ_Contact(in1 := "MODE SELECTION DB"."UF PLC_1 MODE BUFF", in2 := 1)
      { S7_Templates := "SrcType := Int" } EQ_Contact(in1 := "MODE SELECTION DB"."UF PLC_1 PROCESS BUFF", in2 := 495)
      { S7_Templates := "time_type := Time" } "IEC_Timer_0_DB_65".TON(pt := T#5S, et =>)
      Move(in := 500, out1 => "MODE SELECTION DB"."UF PLC_1 PROCESS BUFF")
   END_RUNG
   // the same network as SCL:
   "IEC_Timer_0_DB_65".TON(IN := ("MODE SELECTION DB"."UF PLC_1 MODE BUFF" = 1) AND ("MODE SELECTION DB"."UF PLC_1 PROCESS BUFF" = 495),
                           PT := T#5S);
   IF "IEC_Timer_0_DB_65".Q THEN "MODE SELECTION DB"."UF PLC_1 PROCESS BUFF" := 500; END_IF;
END_REGION

REGION Network 33: SOAK
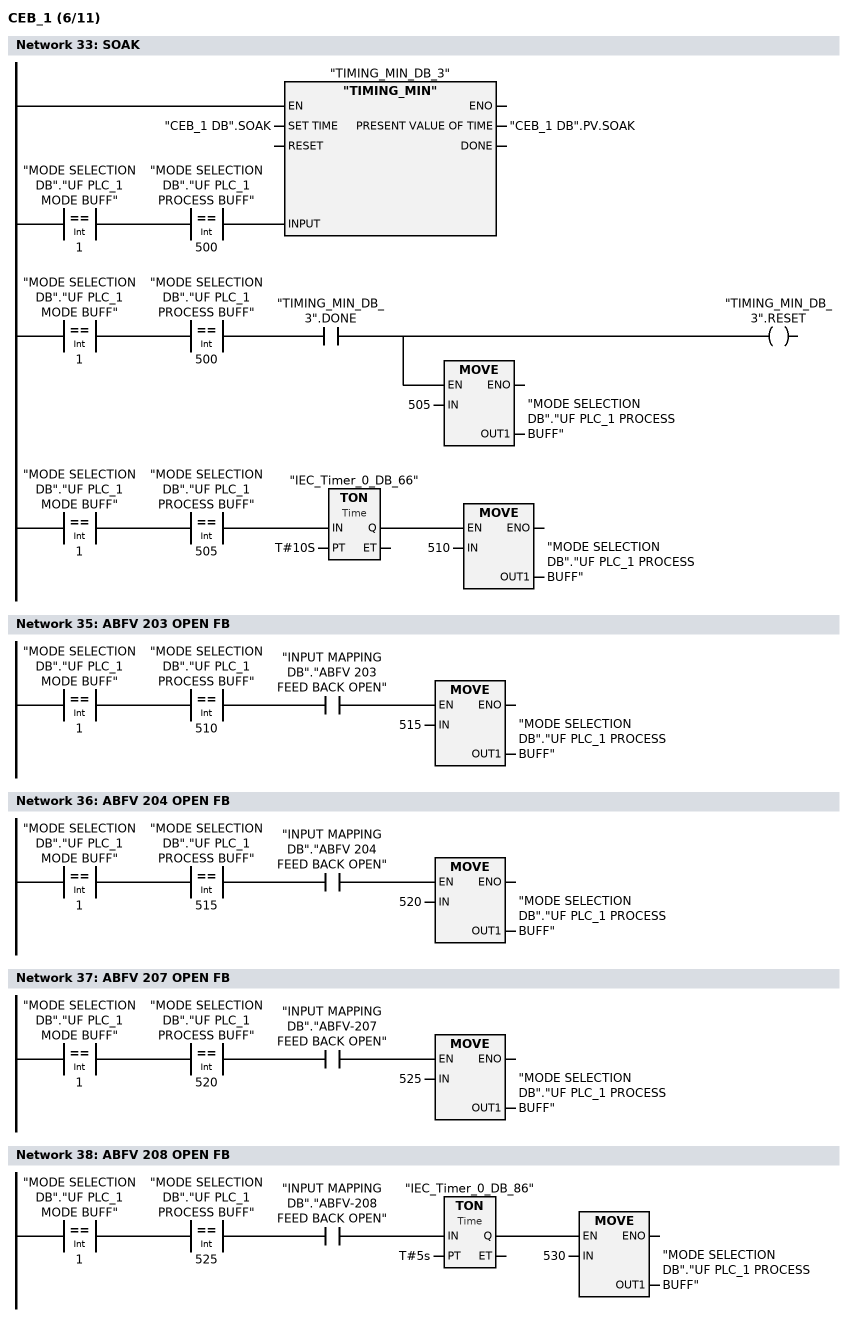
   RUNG wire#powerrail
      "TIMING_MIN_DB_3"(INPUT := wire#w1, "SET TIME" := "CEB_1 DB".SOAK, RESET :=, "PRESENT VALUE OF TIME" => "CEB_1 DB".PV.SOAK, DONE =>)
   END_RUNG
   RUNG wire#powerrail
      { S7_Templates := "SrcType := Int" } EQ_Contact(in1 := "MODE SELECTION DB"."UF PLC_1 MODE BUFF", in2 := 1)
      { S7_Templates := "SrcType := Int" } EQ_Contact(in1 := "MODE SELECTION DB"."UF PLC_1 PROCESS BUFF", in2 := 500)
   END_RUNG wire#w1
   RUNG wire#powerrail
      { S7_Templates := "SrcType := Int" } EQ_Contact(in1 := "MODE SELECTION DB"."UF PLC_1 MODE BUFF", in2 := 1)
      { S7_Templates := "SrcType := Int" } EQ_Contact(in1 := "MODE SELECTION DB"."UF PLC_1 PROCESS BUFF", in2 := 500)
      Contact( "TIMING_MIN_DB_3".DONE )
      wire#w2
      Coil( "TIMING_MIN_DB_3".RESET )
   END_RUNG
   RUNG wire#w2
      Move(in := 505, out1 => "MODE SELECTION DB"."UF PLC_1 PROCESS BUFF")
   END_RUNG
   RUNG wire#powerrail
      { S7_Templates := "SrcType := Int" } EQ_Contact(in1 := "MODE SELECTION DB"."UF PLC_1 MODE BUFF", in2 := 1)
      { S7_Templates := "SrcType := Int" } EQ_Contact(in1 := "MODE SELECTION DB"."UF PLC_1 PROCESS BUFF", in2 := 505)
      { S7_Templates := "time_type := Time" } "IEC_Timer_0_DB_66".TON(pt := T#10S, et =>)
      Move(in := 510, out1 => "MODE SELECTION DB"."UF PLC_1 PROCESS BUFF")
   END_RUNG
   // the same network as SCL:
   "TIMING_MIN_DB_3"("SET TIME" := "CEB_1 DB".SOAK,   // "TIMING_MIN"
                     INPUT := ("MODE SELECTION DB"."UF PLC_1 MODE BUFF" = 1) AND ("MODE SELECTION DB"."UF PLC_1 PROCESS BUFF" = 500),
                     "PRESENT VALUE OF TIME" => "CEB_1 DB".PV.SOAK);
   "TIMING_MIN_DB_3".RESET := ("MODE SELECTION DB"."UF PLC_1 MODE BUFF" = 1) AND ("MODE SELECTION DB"."UF PLC_1 PROCESS BUFF" = 500) AND "TIMING_MIN_DB_3".DONE;
   IF "TIMING_MIN_DB_3".RESET THEN "MODE SELECTION DB"."UF PLC_1 PROCESS BUFF" := 505; END_IF;
   "IEC_Timer_0_DB_66".TON(IN := ("MODE SELECTION DB"."UF PLC_1 MODE BUFF" = 1) AND ("MODE SELECTION DB"."UF PLC_1 PROCESS BUFF" = 505),
                           PT := T#10S);
   IF "IEC_Timer_0_DB_66".Q THEN "MODE SELECTION DB"."UF PLC_1 PROCESS BUFF" := 510; END_IF;
END_REGION

REGION Network 35: ABFV 203 OPEN FB
   RUNG wire#powerrail
      { S7_Templates := "SrcType := Int" } EQ_Contact(in1 := "MODE SELECTION DB"."UF PLC_1 MODE BUFF", in2 := 1)
      { S7_Templates := "SrcType := Int" } EQ_Contact(in1 := "MODE SELECTION DB"."UF PLC_1 PROCESS BUFF", in2 := 510)
      Contact( "INPUT MAPPING DB"."ABFV 203 FEED BACK OPEN" )
      Move(in := 515, out1 => "MODE SELECTION DB"."UF PLC_1 PROCESS BUFF")
   END_RUNG
   // the same network as SCL:
   IF ("MODE SELECTION DB"."UF PLC_1 MODE BUFF" = 1) AND ("MODE SELECTION DB"."UF PLC_1 PROCESS BUFF" = 510) AND "INPUT MAPPING DB"."ABFV 203 FEED BACK OPEN" THEN
       "MODE SELECTION DB"."UF PLC_1 PROCESS BUFF" := 515;
   END_IF;
END_REGION

REGION Network 36: ABFV 204 OPEN FB
   RUNG wire#powerrail
      { S7_Templates := "SrcType := Int" } EQ_Contact(in1 := "MODE SELECTION DB"."UF PLC_1 MODE BUFF", in2 := 1)
      { S7_Templates := "SrcType := Int" } EQ_Contact(in1 := "MODE SELECTION DB"."UF PLC_1 PROCESS BUFF", in2 := 515)
      Contact( "INPUT MAPPING DB"."ABFV 204 FEED BACK OPEN" )
      Move(in := 520, out1 => "MODE SELECTION DB"."UF PLC_1 PROCESS BUFF")
   END_RUNG
   // the same network as SCL:
   IF ("MODE SELECTION DB"."UF PLC_1 MODE BUFF" = 1) AND ("MODE SELECTION DB"."UF PLC_1 PROCESS BUFF" = 515) AND "INPUT MAPPING DB"."ABFV 204 FEED BACK OPEN" THEN
       "MODE SELECTION DB"."UF PLC_1 PROCESS BUFF" := 520;
   END_IF;
END_REGION

REGION Network 37: ABFV 207 OPEN FB
   RUNG wire#powerrail
      { S7_Templates := "SrcType := Int" } EQ_Contact(in1 := "MODE SELECTION DB"."UF PLC_1 MODE BUFF", in2 := 1)
      { S7_Templates := "SrcType := Int" } EQ_Contact(in1 := "MODE SELECTION DB"."UF PLC_1 PROCESS BUFF", in2 := 520)
      Contact( "INPUT MAPPING DB"."ABFV-207 FEED BACK OPEN" )
      Move(in := 525, out1 => "MODE SELECTION DB"."UF PLC_1 PROCESS BUFF")
   END_RUNG
   // the same network as SCL:
   IF ("MODE SELECTION DB"."UF PLC_1 MODE BUFF" = 1) AND ("MODE SELECTION DB"."UF PLC_1 PROCESS BUFF" = 520) AND "INPUT MAPPING DB"."ABFV-207 FEED BACK OPEN" THEN
       "MODE SELECTION DB"."UF PLC_1 PROCESS BUFF" := 525;
   END_IF;
END_REGION

REGION Network 38: ABFV 208 OPEN FB
   RUNG wire#powerrail
      { S7_Templates := "SrcType := Int" } EQ_Contact(in1 := "MODE SELECTION DB"."UF PLC_1 MODE BUFF", in2 := 1)
      { S7_Templates := "SrcType := Int" } EQ_Contact(in1 := "MODE SELECTION DB"."UF PLC_1 PROCESS BUFF", in2 := 525)
      Contact( "INPUT MAPPING DB"."ABFV-208 FEED BACK OPEN" )
      { S7_Templates := "time_type := Time" } "IEC_Timer_0_DB_86".TON(pt := T#5s, et =>)
      Move(in := 530, out1 => "MODE SELECTION DB"."UF PLC_1 PROCESS BUFF")
   END_RUNG
   // the same network as SCL:
   "IEC_Timer_0_DB_86".TON(IN := ("MODE SELECTION DB"."UF PLC_1 MODE BUFF" = 1) AND ("MODE SELECTION DB"."UF PLC_1 PROCESS BUFF" = 525) AND "INPUT MAPPING DB"."ABFV-208 FEED BACK OPEN",
                           PT := T#5s);
   IF "IEC_Timer_0_DB_86".Q THEN "MODE SELECTION DB"."UF PLC_1 PROCESS BUFF" := 530; END_IF;
END_REGION

REGION Network 39: BACKWASH_1
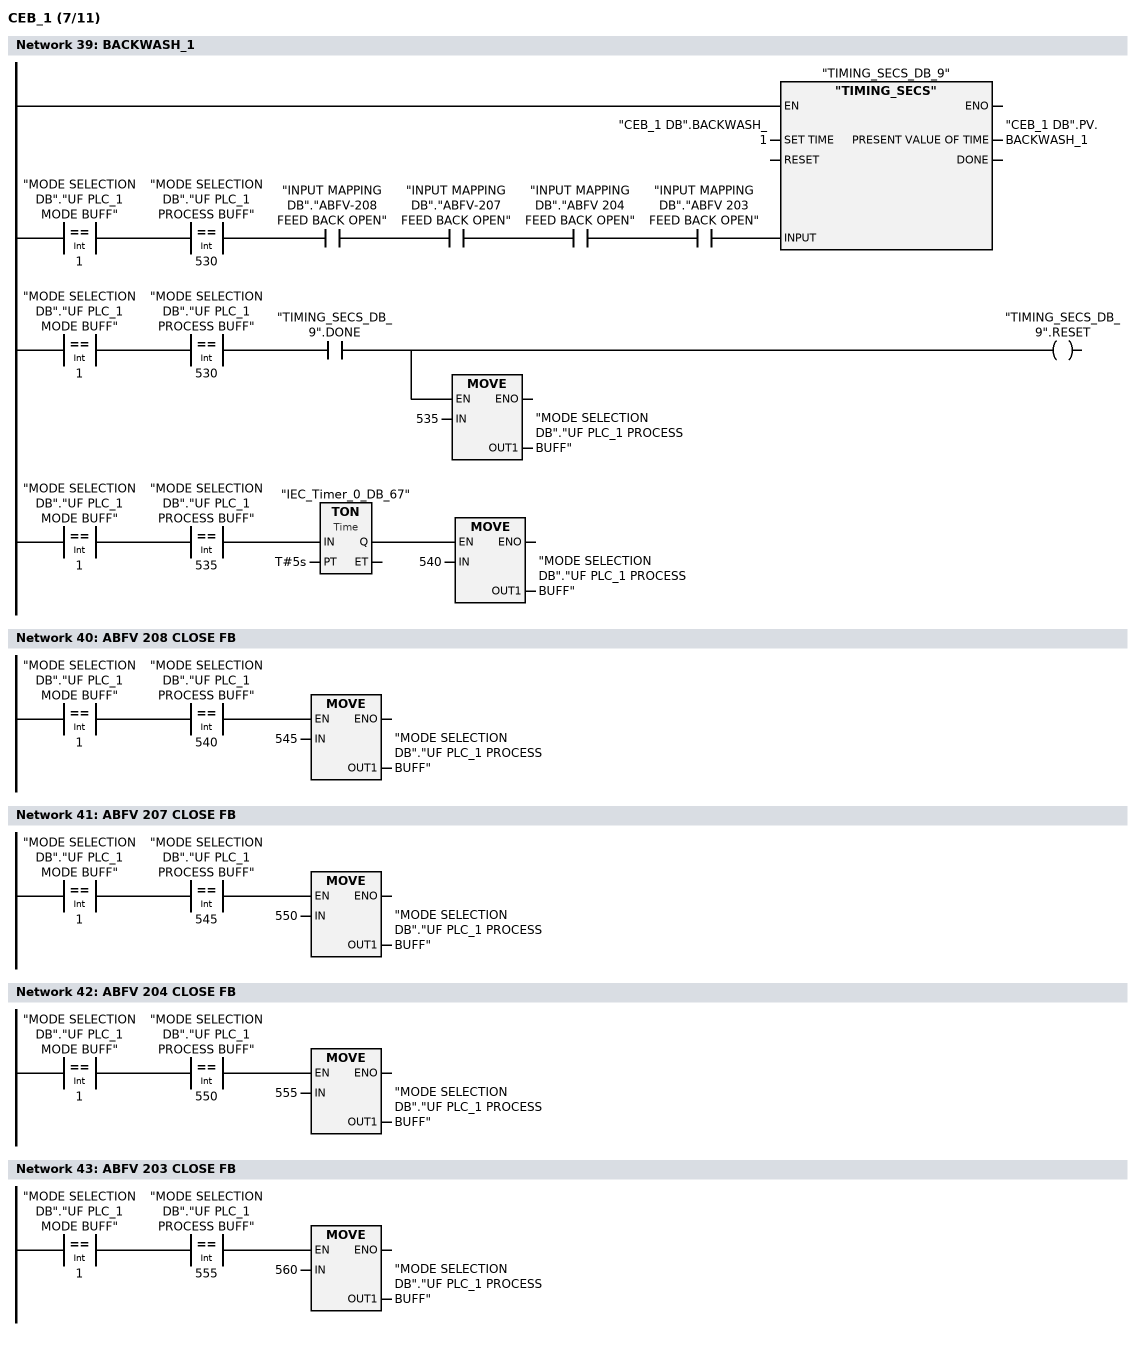
   RUNG wire#powerrail
      "TIMING_SECS_DB_9"(INPUT := wire#w1, "SET TIME" := "CEB_1 DB".BACKWASH_1, RESET :=, "PRESENT VALUE OF TIME" => "CEB_1 DB".PV.BACKWASH_1, DONE =>)
   END_RUNG
   RUNG wire#powerrail
      { S7_Templates := "SrcType := Int" } EQ_Contact(in1 := "MODE SELECTION DB"."UF PLC_1 MODE BUFF", in2 := 1)
      { S7_Templates := "SrcType := Int" } EQ_Contact(in1 := "MODE SELECTION DB"."UF PLC_1 PROCESS BUFF", in2 := 530)
      Contact( "INPUT MAPPING DB"."ABFV-208 FEED BACK OPEN" )
      Contact( "INPUT MAPPING DB"."ABFV-207 FEED BACK OPEN" )
      Contact( "INPUT MAPPING DB"."ABFV 204 FEED BACK OPEN" )
      Contact( "INPUT MAPPING DB"."ABFV 203 FEED BACK OPEN" )
   END_RUNG wire#w1
   RUNG wire#powerrail
      { S7_Templates := "SrcType := Int" } EQ_Contact(in1 := "MODE SELECTION DB"."UF PLC_1 MODE BUFF", in2 := 1)
      { S7_Templates := "SrcType := Int" } EQ_Contact(in1 := "MODE SELECTION DB"."UF PLC_1 PROCESS BUFF", in2 := 530)
      Contact( "TIMING_SECS_DB_9".DONE )
      wire#w2
      Coil( "TIMING_SECS_DB_9".RESET )
   END_RUNG
   RUNG wire#w2
      Move(in := 535, out1 => "MODE SELECTION DB"."UF PLC_1 PROCESS BUFF")
   END_RUNG
   RUNG wire#powerrail
      { S7_Templates := "SrcType := Int" } EQ_Contact(in1 := "MODE SELECTION DB"."UF PLC_1 MODE BUFF", in2 := 1)
      { S7_Templates := "SrcType := Int" } EQ_Contact(in1 := "MODE SELECTION DB"."UF PLC_1 PROCESS BUFF", in2 := 535)
      { S7_Templates := "time_type := Time" } "IEC_Timer_0_DB_67".TON(pt := T#5s, et =>)
      Move(in := 540, out1 => "MODE SELECTION DB"."UF PLC_1 PROCESS BUFF")
   END_RUNG
   // the same network as SCL:
   "TIMING_SECS_DB_9"("SET TIME" := "CEB_1 DB".BACKWASH_1,   // "TIMING_SECS"
                      INPUT := ("MODE SELECTION DB"."UF PLC_1 MODE BUFF" = 1) AND ("MODE SELECTION DB"."UF PLC_1 PROCESS BUFF" = 530) AND "INPUT MAPPING DB"."ABFV-208 FEED BACK OPEN" AND "INPUT MAPPING DB"."ABFV-207 FEED BACK OPEN" AND "INPUT MAPPING DB"."ABFV 204 FEED BACK OPEN" AND "INPUT MAPPING DB"."ABFV 203 FEED BACK OPEN",
                      "PRESENT VALUE OF TIME" => "CEB_1 DB".PV.BACKWASH_1);
   "TIMING_SECS_DB_9".RESET := ("MODE SELECTION DB"."UF PLC_1 MODE BUFF" = 1) AND ("MODE SELECTION DB"."UF PLC_1 PROCESS BUFF" = 530) AND "TIMING_SECS_DB_9".DONE;
   IF "TIMING_SECS_DB_9".RESET THEN "MODE SELECTION DB"."UF PLC_1 PROCESS BUFF" := 535; END_IF;
   "IEC_Timer_0_DB_67".TON(IN := ("MODE SELECTION DB"."UF PLC_1 MODE BUFF" = 1) AND ("MODE SELECTION DB"."UF PLC_1 PROCESS BUFF" = 535),
                           PT := T#5s);
   IF "IEC_Timer_0_DB_67".Q THEN "MODE SELECTION DB"."UF PLC_1 PROCESS BUFF" := 540; END_IF;
END_REGION

REGION Network 40: ABFV 208 CLOSE FB
   RUNG wire#powerrail
      { S7_Templates := "SrcType := Int" } EQ_Contact(in1 := "MODE SELECTION DB"."UF PLC_1 MODE BUFF", in2 := 1)
      { S7_Templates := "SrcType := Int" } EQ_Contact(in1 := "MODE SELECTION DB"."UF PLC_1 PROCESS BUFF", in2 := 540)
      Move(in := 545, out1 => "MODE SELECTION DB"."UF PLC_1 PROCESS BUFF")
   END_RUNG
   // the same network as SCL:
   IF ("MODE SELECTION DB"."UF PLC_1 MODE BUFF" = 1) AND ("MODE SELECTION DB"."UF PLC_1 PROCESS BUFF" = 540) THEN
       "MODE SELECTION DB"."UF PLC_1 PROCESS BUFF" := 545;
   END_IF;
END_REGION

REGION Network 41: ABFV 207 CLOSE FB
   RUNG wire#powerrail
      { S7_Templates := "SrcType := Int" } EQ_Contact(in1 := "MODE SELECTION DB"."UF PLC_1 MODE BUFF", in2 := 1)
      { S7_Templates := "SrcType := Int" } EQ_Contact(in1 := "MODE SELECTION DB"."UF PLC_1 PROCESS BUFF", in2 := 545)
      Move(in := 550, out1 => "MODE SELECTION DB"."UF PLC_1 PROCESS BUFF")
   END_RUNG
   // the same network as SCL:
   IF ("MODE SELECTION DB"."UF PLC_1 MODE BUFF" = 1) AND ("MODE SELECTION DB"."UF PLC_1 PROCESS BUFF" = 545) THEN
       "MODE SELECTION DB"."UF PLC_1 PROCESS BUFF" := 550;
   END_IF;
END_REGION

REGION Network 42: ABFV 204 CLOSE FB
   RUNG wire#powerrail
      { S7_Templates := "SrcType := Int" } EQ_Contact(in1 := "MODE SELECTION DB"."UF PLC_1 MODE BUFF", in2 := 1)
      { S7_Templates := "SrcType := Int" } EQ_Contact(in1 := "MODE SELECTION DB"."UF PLC_1 PROCESS BUFF", in2 := 550)
      Move(in := 555, out1 => "MODE SELECTION DB"."UF PLC_1 PROCESS BUFF")
   END_RUNG
   // the same network as SCL:
   IF ("MODE SELECTION DB"."UF PLC_1 MODE BUFF" = 1) AND ("MODE SELECTION DB"."UF PLC_1 PROCESS BUFF" = 550) THEN
       "MODE SELECTION DB"."UF PLC_1 PROCESS BUFF" := 555;
   END_IF;
END_REGION

REGION Network 43: ABFV 203 CLOSE FB
   RUNG wire#powerrail
      { S7_Templates := "SrcType := Int" } EQ_Contact(in1 := "MODE SELECTION DB"."UF PLC_1 MODE BUFF", in2 := 1)
      { S7_Templates := "SrcType := Int" } EQ_Contact(in1 := "MODE SELECTION DB"."UF PLC_1 PROCESS BUFF", in2 := 555)
      Move(in := 560, out1 => "MODE SELECTION DB"."UF PLC_1 PROCESS BUFF")
   END_RUNG
   // the same network as SCL:
   IF ("MODE SELECTION DB"."UF PLC_1 MODE BUFF" = 1) AND ("MODE SELECTION DB"."UF PLC_1 PROCESS BUFF" = 555) THEN
       "MODE SELECTION DB"."UF PLC_1 PROCESS BUFF" := 560;
   END_IF;
END_REGION

REGION Network 44: 565
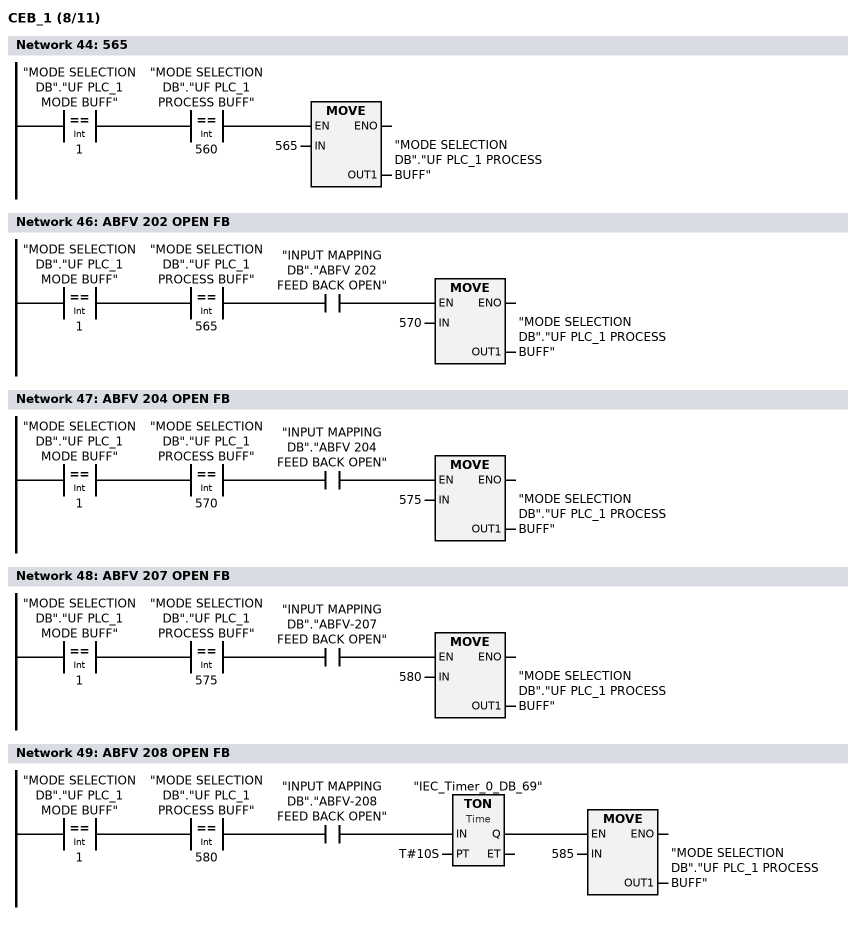
   RUNG wire#powerrail
      { S7_Templates := "SrcType := Int" } EQ_Contact(in1 := "MODE SELECTION DB"."UF PLC_1 MODE BUFF", in2 := 1)
      { S7_Templates := "SrcType := Int" } EQ_Contact(in1 := "MODE SELECTION DB"."UF PLC_1 PROCESS BUFF", in2 := 560)
      Move(in := 565, out1 => "MODE SELECTION DB"."UF PLC_1 PROCESS BUFF")
   END_RUNG
   // the same network as SCL:
   IF ("MODE SELECTION DB"."UF PLC_1 MODE BUFF" = 1) AND ("MODE SELECTION DB"."UF PLC_1 PROCESS BUFF" = 560) THEN
       "MODE SELECTION DB"."UF PLC_1 PROCESS BUFF" := 565;
   END_IF;
END_REGION

REGION Network 46: ABFV 202 OPEN FB
   RUNG wire#powerrail
      { S7_Templates := "SrcType := Int" } EQ_Contact(in1 := "MODE SELECTION DB"."UF PLC_1 MODE BUFF", in2 := 1)
      { S7_Templates := "SrcType := Int" } EQ_Contact(in1 := "MODE SELECTION DB"."UF PLC_1 PROCESS BUFF", in2 := 565)
      Contact( "INPUT MAPPING DB"."ABFV 202 FEED BACK OPEN" )
      Move(in := 570, out1 => "MODE SELECTION DB"."UF PLC_1 PROCESS BUFF")
   END_RUNG
   // the same network as SCL:
   IF ("MODE SELECTION DB"."UF PLC_1 MODE BUFF" = 1) AND ("MODE SELECTION DB"."UF PLC_1 PROCESS BUFF" = 565) AND "INPUT MAPPING DB"."ABFV 202 FEED BACK OPEN" THEN
       "MODE SELECTION DB"."UF PLC_1 PROCESS BUFF" := 570;
   END_IF;
END_REGION

REGION Network 47: ABFV 204 OPEN FB
   RUNG wire#powerrail
      { S7_Templates := "SrcType := Int" } EQ_Contact(in1 := "MODE SELECTION DB"."UF PLC_1 MODE BUFF", in2 := 1)
      { S7_Templates := "SrcType := Int" } EQ_Contact(in1 := "MODE SELECTION DB"."UF PLC_1 PROCESS BUFF", in2 := 570)
      Contact( "INPUT MAPPING DB"."ABFV 204 FEED BACK OPEN" )
      Move(in := 575, out1 => "MODE SELECTION DB"."UF PLC_1 PROCESS BUFF")
   END_RUNG
   // the same network as SCL:
   IF ("MODE SELECTION DB"."UF PLC_1 MODE BUFF" = 1) AND ("MODE SELECTION DB"."UF PLC_1 PROCESS BUFF" = 570) AND "INPUT MAPPING DB"."ABFV 204 FEED BACK OPEN" THEN
       "MODE SELECTION DB"."UF PLC_1 PROCESS BUFF" := 575;
   END_IF;
END_REGION

REGION Network 48: ABFV 207 OPEN FB
   RUNG wire#powerrail
      { S7_Templates := "SrcType := Int" } EQ_Contact(in1 := "MODE SELECTION DB"."UF PLC_1 MODE BUFF", in2 := 1)
      { S7_Templates := "SrcType := Int" } EQ_Contact(in1 := "MODE SELECTION DB"."UF PLC_1 PROCESS BUFF", in2 := 575)
      Contact( "INPUT MAPPING DB"."ABFV-207 FEED BACK OPEN" )
      Move(in := 580, out1 => "MODE SELECTION DB"."UF PLC_1 PROCESS BUFF")
   END_RUNG
   // the same network as SCL:
   IF ("MODE SELECTION DB"."UF PLC_1 MODE BUFF" = 1) AND ("MODE SELECTION DB"."UF PLC_1 PROCESS BUFF" = 575) AND "INPUT MAPPING DB"."ABFV-207 FEED BACK OPEN" THEN
       "MODE SELECTION DB"."UF PLC_1 PROCESS BUFF" := 580;
   END_IF;
END_REGION

REGION Network 49: ABFV 208 OPEN FB
   RUNG wire#powerrail
      { S7_Templates := "SrcType := Int" } EQ_Contact(in1 := "MODE SELECTION DB"."UF PLC_1 MODE BUFF", in2 := 1)
      { S7_Templates := "SrcType := Int" } EQ_Contact(in1 := "MODE SELECTION DB"."UF PLC_1 PROCESS BUFF", in2 := 580)
      Contact( "INPUT MAPPING DB"."ABFV-208 FEED BACK OPEN" )
      { S7_Templates := "time_type := Time" } "IEC_Timer_0_DB_69".TON(pt := T#10S, et =>)
      Move(in := 585, out1 => "MODE SELECTION DB"."UF PLC_1 PROCESS BUFF")
   END_RUNG
   // the same network as SCL:
   "IEC_Timer_0_DB_69".TON(IN := ("MODE SELECTION DB"."UF PLC_1 MODE BUFF" = 1) AND ("MODE SELECTION DB"."UF PLC_1 PROCESS BUFF" = 580) AND "INPUT MAPPING DB"."ABFV-208 FEED BACK OPEN",
                           PT := T#10S);
   IF "IEC_Timer_0_DB_69".Q THEN "MODE SELECTION DB"."UF PLC_1 PROCESS BUFF" := 585; END_IF;
END_REGION

REGION Network 50: BACKWASH_2
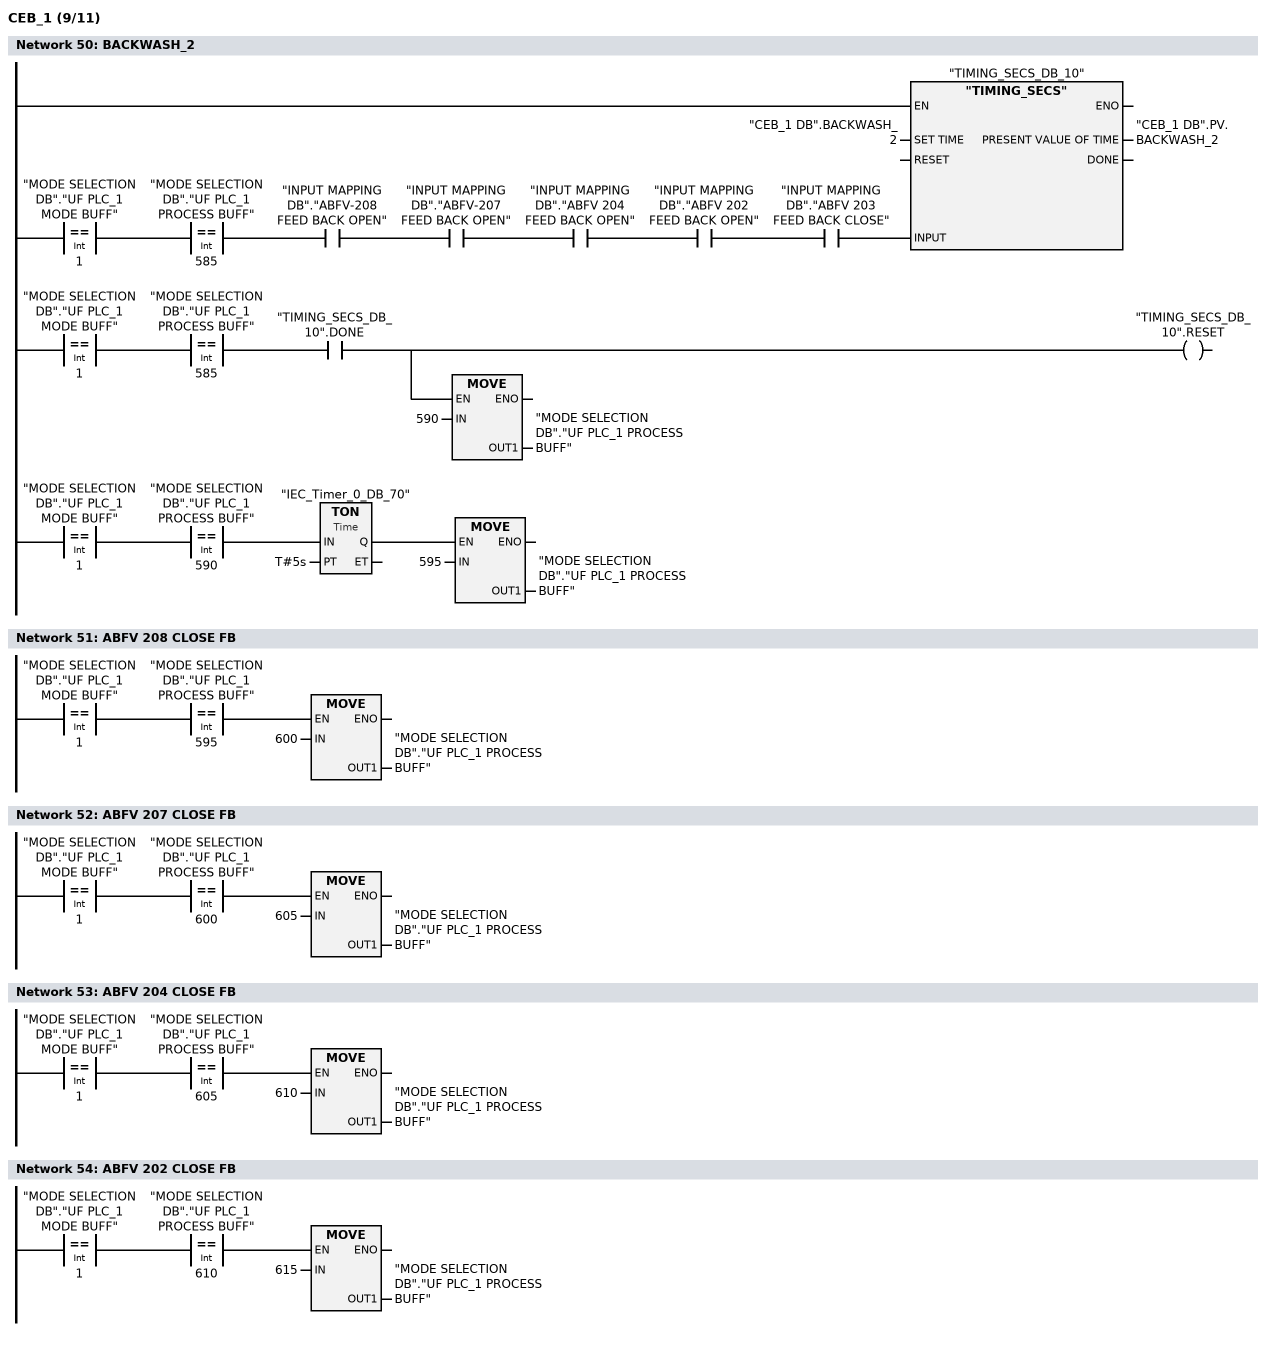
   RUNG wire#powerrail
      "TIMING_SECS_DB_10"(INPUT := wire#w1, "SET TIME" := "CEB_1 DB".BACKWASH_2, RESET :=, "PRESENT VALUE OF TIME" => "CEB_1 DB".PV.BACKWASH_2, DONE =>)
   END_RUNG
   RUNG wire#powerrail
      { S7_Templates := "SrcType := Int" } EQ_Contact(in1 := "MODE SELECTION DB"."UF PLC_1 MODE BUFF", in2 := 1)
      { S7_Templates := "SrcType := Int" } EQ_Contact(in1 := "MODE SELECTION DB"."UF PLC_1 PROCESS BUFF", in2 := 585)
      Contact( "INPUT MAPPING DB"."ABFV-208 FEED BACK OPEN" )
      Contact( "INPUT MAPPING DB"."ABFV-207 FEED BACK OPEN" )
      Contact( "INPUT MAPPING DB"."ABFV 204 FEED BACK OPEN" )
      Contact( "INPUT MAPPING DB"."ABFV 202 FEED BACK OPEN" )
      Contact( "INPUT MAPPING DB"."ABFV 203 FEED BACK CLOSE" )
   END_RUNG wire#w1
   RUNG wire#powerrail
      { S7_Templates := "SrcType := Int" } EQ_Contact(in1 := "MODE SELECTION DB"."UF PLC_1 MODE BUFF", in2 := 1)
      { S7_Templates := "SrcType := Int" } EQ_Contact(in1 := "MODE SELECTION DB"."UF PLC_1 PROCESS BUFF", in2 := 585)
      Contact( "TIMING_SECS_DB_10".DONE )
      wire#w2
      Coil( "TIMING_SECS_DB_10".RESET )
   END_RUNG
   RUNG wire#w2
      Move(in := 590, out1 => "MODE SELECTION DB"."UF PLC_1 PROCESS BUFF")
   END_RUNG
   RUNG wire#powerrail
      { S7_Templates := "SrcType := Int" } EQ_Contact(in1 := "MODE SELECTION DB"."UF PLC_1 MODE BUFF", in2 := 1)
      { S7_Templates := "SrcType := Int" } EQ_Contact(in1 := "MODE SELECTION DB"."UF PLC_1 PROCESS BUFF", in2 := 590)
      { S7_Templates := "time_type := Time" } "IEC_Timer_0_DB_70".TON(pt := T#5s, et =>)
      Move(in := 595, out1 => "MODE SELECTION DB"."UF PLC_1 PROCESS BUFF")
   END_RUNG
   // the same network as SCL:
   "TIMING_SECS_DB_10"("SET TIME" := "CEB_1 DB".BACKWASH_2,   // "TIMING_SECS"
                       INPUT := ("MODE SELECTION DB"."UF PLC_1 MODE BUFF" = 1) AND ("MODE SELECTION DB"."UF PLC_1 PROCESS BUFF" = 585) AND "INPUT MAPPING DB"."ABFV-208 FEED BACK OPEN" AND "INPUT MAPPING DB"."ABFV-207 FEED BACK OPEN" AND "INPUT MAPPING DB"."ABFV 204 FEED BACK OPEN" AND "INPUT MAPPING DB"."ABFV 202 FEED BACK OPEN" AND "INPUT MAPPING DB"."ABFV 203 FEED BACK CLOSE",
                       "PRESENT VALUE OF TIME" => "CEB_1 DB".PV.BACKWASH_2);
   "TIMING_SECS_DB_10".RESET := ("MODE SELECTION DB"."UF PLC_1 MODE BUFF" = 1) AND ("MODE SELECTION DB"."UF PLC_1 PROCESS BUFF" = 585) AND "TIMING_SECS_DB_10".DONE;
   IF "TIMING_SECS_DB_10".RESET THEN "MODE SELECTION DB"."UF PLC_1 PROCESS BUFF" := 590; END_IF;
   "IEC_Timer_0_DB_70".TON(IN := ("MODE SELECTION DB"."UF PLC_1 MODE BUFF" = 1) AND ("MODE SELECTION DB"."UF PLC_1 PROCESS BUFF" = 590),
                           PT := T#5s);
   IF "IEC_Timer_0_DB_70".Q THEN "MODE SELECTION DB"."UF PLC_1 PROCESS BUFF" := 595; END_IF;
END_REGION

REGION Network 51: ABFV 208 CLOSE FB
   RUNG wire#powerrail
      { S7_Templates := "SrcType := Int" } EQ_Contact(in1 := "MODE SELECTION DB"."UF PLC_1 MODE BUFF", in2 := 1)
      { S7_Templates := "SrcType := Int" } EQ_Contact(in1 := "MODE SELECTION DB"."UF PLC_1 PROCESS BUFF", in2 := 595)
      Move(in := 600, out1 => "MODE SELECTION DB"."UF PLC_1 PROCESS BUFF")
   END_RUNG
   // the same network as SCL:
   IF ("MODE SELECTION DB"."UF PLC_1 MODE BUFF" = 1) AND ("MODE SELECTION DB"."UF PLC_1 PROCESS BUFF" = 595) THEN
       "MODE SELECTION DB"."UF PLC_1 PROCESS BUFF" := 600;
   END_IF;
END_REGION

REGION Network 52: ABFV 207 CLOSE FB
   RUNG wire#powerrail
      { S7_Templates := "SrcType := Int" } EQ_Contact(in1 := "MODE SELECTION DB"."UF PLC_1 MODE BUFF", in2 := 1)
      { S7_Templates := "SrcType := Int" } EQ_Contact(in1 := "MODE SELECTION DB"."UF PLC_1 PROCESS BUFF", in2 := 600)
      Move(in := 605, out1 => "MODE SELECTION DB"."UF PLC_1 PROCESS BUFF")
   END_RUNG
   // the same network as SCL:
   IF ("MODE SELECTION DB"."UF PLC_1 MODE BUFF" = 1) AND ("MODE SELECTION DB"."UF PLC_1 PROCESS BUFF" = 600) THEN
       "MODE SELECTION DB"."UF PLC_1 PROCESS BUFF" := 605;
   END_IF;
END_REGION

REGION Network 53: ABFV 204 CLOSE FB
   RUNG wire#powerrail
      { S7_Templates := "SrcType := Int" } EQ_Contact(in1 := "MODE SELECTION DB"."UF PLC_1 MODE BUFF", in2 := 1)
      { S7_Templates := "SrcType := Int" } EQ_Contact(in1 := "MODE SELECTION DB"."UF PLC_1 PROCESS BUFF", in2 := 605)
      Move(in := 610, out1 => "MODE SELECTION DB"."UF PLC_1 PROCESS BUFF")
   END_RUNG
   // the same network as SCL:
   IF ("MODE SELECTION DB"."UF PLC_1 MODE BUFF" = 1) AND ("MODE SELECTION DB"."UF PLC_1 PROCESS BUFF" = 605) THEN
       "MODE SELECTION DB"."UF PLC_1 PROCESS BUFF" := 610;
   END_IF;
END_REGION

REGION Network 54: ABFV 202 CLOSE FB
   RUNG wire#powerrail
      { S7_Templates := "SrcType := Int" } EQ_Contact(in1 := "MODE SELECTION DB"."UF PLC_1 MODE BUFF", in2 := 1)
      { S7_Templates := "SrcType := Int" } EQ_Contact(in1 := "MODE SELECTION DB"."UF PLC_1 PROCESS BUFF", in2 := 610)
      Move(in := 615, out1 => "MODE SELECTION DB"."UF PLC_1 PROCESS BUFF")
   END_RUNG
   // the same network as SCL:
   IF ("MODE SELECTION DB"."UF PLC_1 MODE BUFF" = 1) AND ("MODE SELECTION DB"."UF PLC_1 PROCESS BUFF" = 610) THEN
       "MODE SELECTION DB"."UF PLC_1 PROCESS BUFF" := 615;
   END_IF;
END_REGION

REGION Network 55: 620
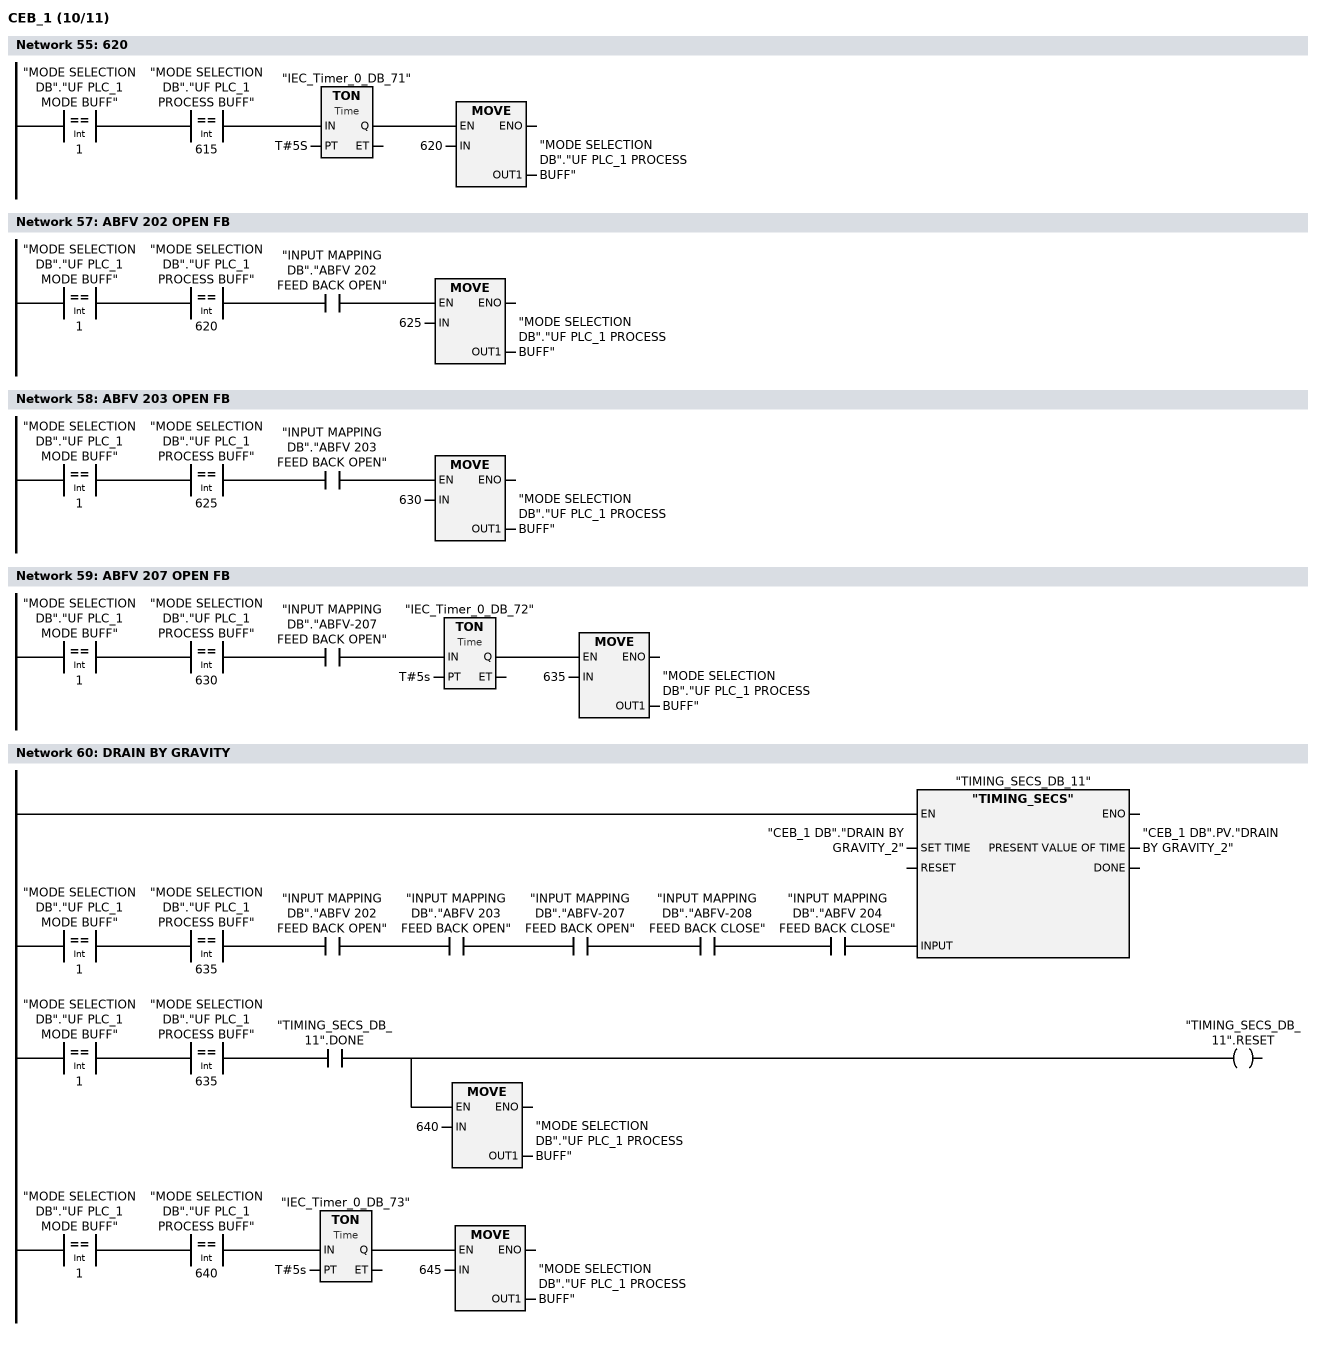
   RUNG wire#powerrail
      { S7_Templates := "SrcType := Int" } EQ_Contact(in1 := "MODE SELECTION DB"."UF PLC_1 MODE BUFF", in2 := 1)
      { S7_Templates := "SrcType := Int" } EQ_Contact(in1 := "MODE SELECTION DB"."UF PLC_1 PROCESS BUFF", in2 := 615)
      { S7_Templates := "time_type := Time" } "IEC_Timer_0_DB_71".TON(pt := T#5S, et =>)
      Move(in := 620, out1 => "MODE SELECTION DB"."UF PLC_1 PROCESS BUFF")
   END_RUNG
   // the same network as SCL:
   "IEC_Timer_0_DB_71".TON(IN := ("MODE SELECTION DB"."UF PLC_1 MODE BUFF" = 1) AND ("MODE SELECTION DB"."UF PLC_1 PROCESS BUFF" = 615),
                           PT := T#5S);
   IF "IEC_Timer_0_DB_71".Q THEN "MODE SELECTION DB"."UF PLC_1 PROCESS BUFF" := 620; END_IF;
END_REGION

REGION Network 57: ABFV 202 OPEN FB
   RUNG wire#powerrail
      { S7_Templates := "SrcType := Int" } EQ_Contact(in1 := "MODE SELECTION DB"."UF PLC_1 MODE BUFF", in2 := 1)
      { S7_Templates := "SrcType := Int" } EQ_Contact(in1 := "MODE SELECTION DB"."UF PLC_1 PROCESS BUFF", in2 := 620)
      Contact( "INPUT MAPPING DB"."ABFV 202 FEED BACK OPEN" )
      Move(in := 625, out1 => "MODE SELECTION DB"."UF PLC_1 PROCESS BUFF")
   END_RUNG
   // the same network as SCL:
   IF ("MODE SELECTION DB"."UF PLC_1 MODE BUFF" = 1) AND ("MODE SELECTION DB"."UF PLC_1 PROCESS BUFF" = 620) AND "INPUT MAPPING DB"."ABFV 202 FEED BACK OPEN" THEN
       "MODE SELECTION DB"."UF PLC_1 PROCESS BUFF" := 625;
   END_IF;
END_REGION

REGION Network 58: ABFV 203 OPEN FB
   RUNG wire#powerrail
      { S7_Templates := "SrcType := Int" } EQ_Contact(in1 := "MODE SELECTION DB"."UF PLC_1 MODE BUFF", in2 := 1)
      { S7_Templates := "SrcType := Int" } EQ_Contact(in1 := "MODE SELECTION DB"."UF PLC_1 PROCESS BUFF", in2 := 625)
      Contact( "INPUT MAPPING DB"."ABFV 203 FEED BACK OPEN" )
      Move(in := 630, out1 => "MODE SELECTION DB"."UF PLC_1 PROCESS BUFF")
   END_RUNG
   // the same network as SCL:
   IF ("MODE SELECTION DB"."UF PLC_1 MODE BUFF" = 1) AND ("MODE SELECTION DB"."UF PLC_1 PROCESS BUFF" = 625) AND "INPUT MAPPING DB"."ABFV 203 FEED BACK OPEN" THEN
       "MODE SELECTION DB"."UF PLC_1 PROCESS BUFF" := 630;
   END_IF;
END_REGION

REGION Network 59: ABFV 207 OPEN FB
   RUNG wire#powerrail
      { S7_Templates := "SrcType := Int" } EQ_Contact(in1 := "MODE SELECTION DB"."UF PLC_1 MODE BUFF", in2 := 1)
      { S7_Templates := "SrcType := Int" } EQ_Contact(in1 := "MODE SELECTION DB"."UF PLC_1 PROCESS BUFF", in2 := 630)
      Contact( "INPUT MAPPING DB"."ABFV-207 FEED BACK OPEN" )
      { S7_Templates := "time_type := Time" } "IEC_Timer_0_DB_72".TON(pt := T#5s, et =>)
      Move(in := 635, out1 => "MODE SELECTION DB"."UF PLC_1 PROCESS BUFF")
   END_RUNG
   // the same network as SCL:
   "IEC_Timer_0_DB_72".TON(IN := ("MODE SELECTION DB"."UF PLC_1 MODE BUFF" = 1) AND ("MODE SELECTION DB"."UF PLC_1 PROCESS BUFF" = 630) AND "INPUT MAPPING DB"."ABFV-207 FEED BACK OPEN",
                           PT := T#5s);
   IF "IEC_Timer_0_DB_72".Q THEN "MODE SELECTION DB"."UF PLC_1 PROCESS BUFF" := 635; END_IF;
END_REGION

REGION Network 60: DRAIN BY GRAVITY
   RUNG wire#powerrail
      "TIMING_SECS_DB_11"(INPUT := wire#w1, "SET TIME" := "CEB_1 DB"."DRAIN BY GRAVITY_2", RESET :=, "PRESENT VALUE OF TIME" => "CEB_1 DB".PV."DRAIN BY GRAVITY_2", DONE =>)
   END_RUNG
   RUNG wire#powerrail
      { S7_Templates := "SrcType := Int" } EQ_Contact(in1 := "MODE SELECTION DB"."UF PLC_1 MODE BUFF", in2 := 1)
      { S7_Templates := "SrcType := Int" } EQ_Contact(in1 := "MODE SELECTION DB"."UF PLC_1 PROCESS BUFF", in2 := 635)
      Contact( "INPUT MAPPING DB"."ABFV 202 FEED BACK OPEN" )
      Contact( "INPUT MAPPING DB"."ABFV 203 FEED BACK OPEN" )
      Contact( "INPUT MAPPING DB"."ABFV-207 FEED BACK OPEN" )
      Contact( "INPUT MAPPING DB"."ABFV-208 FEED BACK CLOSE" )
      Contact( "INPUT MAPPING DB"."ABFV 204 FEED BACK CLOSE" )
   END_RUNG wire#w1
   RUNG wire#powerrail
      { S7_Templates := "SrcType := Int" } EQ_Contact(in1 := "MODE SELECTION DB"."UF PLC_1 MODE BUFF", in2 := 1)
      { S7_Templates := "SrcType := Int" } EQ_Contact(in1 := "MODE SELECTION DB"."UF PLC_1 PROCESS BUFF", in2 := 635)
      Contact( "TIMING_SECS_DB_11".DONE )
      wire#w2
      Coil( "TIMING_SECS_DB_11".RESET )
   END_RUNG
   RUNG wire#w2
      Move(in := 640, out1 => "MODE SELECTION DB"."UF PLC_1 PROCESS BUFF")
   END_RUNG
   RUNG wire#powerrail
      { S7_Templates := "SrcType := Int" } EQ_Contact(in1 := "MODE SELECTION DB"."UF PLC_1 MODE BUFF", in2 := 1)
      { S7_Templates := "SrcType := Int" } EQ_Contact(in1 := "MODE SELECTION DB"."UF PLC_1 PROCESS BUFF", in2 := 640)
      { S7_Templates := "time_type := Time" } "IEC_Timer_0_DB_73".TON(pt := T#5s, et =>)
      Move(in := 645, out1 => "MODE SELECTION DB"."UF PLC_1 PROCESS BUFF")
   END_RUNG
   // the same network as SCL:
   "TIMING_SECS_DB_11"("SET TIME" := "CEB_1 DB"."DRAIN BY GRAVITY_2",   // "TIMING_SECS"
                       INPUT := ("MODE SELECTION DB"."UF PLC_1 MODE BUFF" = 1) AND ("MODE SELECTION DB"."UF PLC_1 PROCESS BUFF" = 635) AND "INPUT MAPPING DB"."ABFV 202 FEED BACK OPEN" AND "INPUT MAPPING DB"."ABFV 203 FEED BACK OPEN" AND "INPUT MAPPING DB"."ABFV-207 FEED BACK OPEN" AND "INPUT MAPPING DB"."ABFV-208 FEED BACK CLOSE" AND "INPUT MAPPING DB"."ABFV 204 FEED BACK CLOSE",
                       "PRESENT VALUE OF TIME" => "CEB_1 DB".PV."DRAIN BY GRAVITY_2");
   "TIMING_SECS_DB_11".RESET := ("MODE SELECTION DB"."UF PLC_1 MODE BUFF" = 1) AND ("MODE SELECTION DB"."UF PLC_1 PROCESS BUFF" = 635) AND "TIMING_SECS_DB_11".DONE;
   IF "TIMING_SECS_DB_11".RESET THEN "MODE SELECTION DB"."UF PLC_1 PROCESS BUFF" := 640; END_IF;
   "IEC_Timer_0_DB_73".TON(IN := ("MODE SELECTION DB"."UF PLC_1 MODE BUFF" = 1) AND ("MODE SELECTION DB"."UF PLC_1 PROCESS BUFF" = 640),
                           PT := T#5s);
   IF "IEC_Timer_0_DB_73".Q THEN "MODE SELECTION DB"."UF PLC_1 PROCESS BUFF" := 645; END_IF;
END_REGION

REGION Network 61: ABFV 207 CLOSE FB
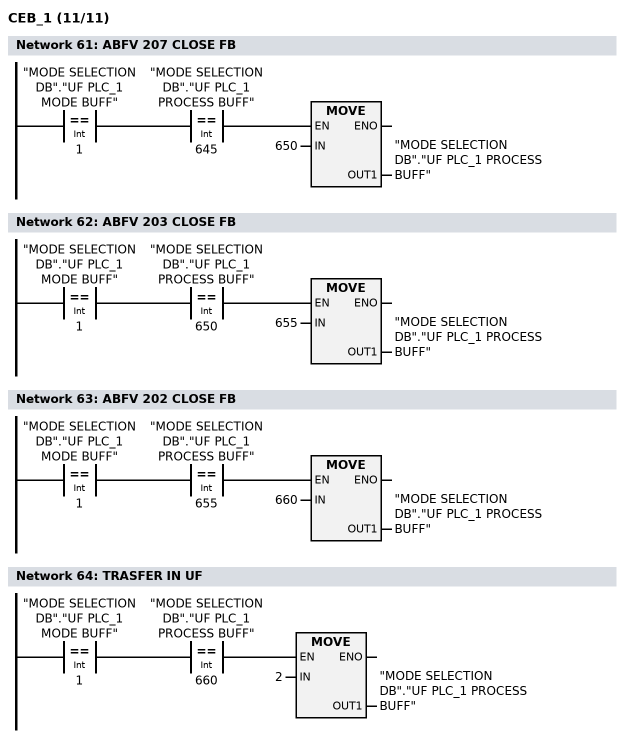
   RUNG wire#powerrail
      { S7_Templates := "SrcType := Int" } EQ_Contact(in1 := "MODE SELECTION DB"."UF PLC_1 MODE BUFF", in2 := 1)
      { S7_Templates := "SrcType := Int" } EQ_Contact(in1 := "MODE SELECTION DB"."UF PLC_1 PROCESS BUFF", in2 := 645)
      Move(in := 650, out1 => "MODE SELECTION DB"."UF PLC_1 PROCESS BUFF")
   END_RUNG
   // the same network as SCL:
   IF ("MODE SELECTION DB"."UF PLC_1 MODE BUFF" = 1) AND ("MODE SELECTION DB"."UF PLC_1 PROCESS BUFF" = 645) THEN
       "MODE SELECTION DB"."UF PLC_1 PROCESS BUFF" := 650;
   END_IF;
END_REGION

REGION Network 62: ABFV 203 CLOSE FB
   RUNG wire#powerrail
      { S7_Templates := "SrcType := Int" } EQ_Contact(in1 := "MODE SELECTION DB"."UF PLC_1 MODE BUFF", in2 := 1)
      { S7_Templates := "SrcType := Int" } EQ_Contact(in1 := "MODE SELECTION DB"."UF PLC_1 PROCESS BUFF", in2 := 650)
      Move(in := 655, out1 => "MODE SELECTION DB"."UF PLC_1 PROCESS BUFF")
   END_RUNG
   // the same network as SCL:
   IF ("MODE SELECTION DB"."UF PLC_1 MODE BUFF" = 1) AND ("MODE SELECTION DB"."UF PLC_1 PROCESS BUFF" = 650) THEN
       "MODE SELECTION DB"."UF PLC_1 PROCESS BUFF" := 655;
   END_IF;
END_REGION

REGION Network 63: ABFV 202 CLOSE FB
   RUNG wire#powerrail
      { S7_Templates := "SrcType := Int" } EQ_Contact(in1 := "MODE SELECTION DB"."UF PLC_1 MODE BUFF", in2 := 1)
      { S7_Templates := "SrcType := Int" } EQ_Contact(in1 := "MODE SELECTION DB"."UF PLC_1 PROCESS BUFF", in2 := 655)
      Move(in := 660, out1 => "MODE SELECTION DB"."UF PLC_1 PROCESS BUFF")
   END_RUNG
   // the same network as SCL:
   IF ("MODE SELECTION DB"."UF PLC_1 MODE BUFF" = 1) AND ("MODE SELECTION DB"."UF PLC_1 PROCESS BUFF" = 655) THEN
       "MODE SELECTION DB"."UF PLC_1 PROCESS BUFF" := 660;
   END_IF;
END_REGION

REGION Network 64: TRASFER IN UF
   RUNG wire#powerrail
      { S7_Templates := "SrcType := Int" } EQ_Contact(in1 := "MODE SELECTION DB"."UF PLC_1 MODE BUFF", in2 := 1)
      { S7_Templates := "SrcType := Int" } EQ_Contact(in1 := "MODE SELECTION DB"."UF PLC_1 PROCESS BUFF", in2 := 660)
      Move(in := 2, out1 => "MODE SELECTION DB"."UF PLC_1 PROCESS BUFF")
   END_RUNG
   // the same network as SCL:
   IF ("MODE SELECTION DB"."UF PLC_1 MODE BUFF" = 1) AND ("MODE SELECTION DB"."UF PLC_1 PROCESS BUFF" = 660) THEN
       "MODE SELECTION DB"."UF PLC_1 PROCESS BUFF" := 2;
   END_IF;
END_REGION
END_FUNCTION
